(* CoDeSys 2.3.9.45 project: Ascenseur_Augustin_FUCHS.pro *)
(* Libraries: standard.lib 2.6.14 10:37:46, Util.lib 26.9.14 10:12:46 *)

(* Global variable list: Variables_Globales *)
VAR_GLOBAL
(* ----------------------------------
	Entrée
-------------------------------------*)
	(*Présence étage*)
	PRDC: BOOL;
	PET1: BOOL;
	PET2: BOOL;
	PET3: BOOL;

	(*Appel à partir du palier de l'étage*)
	PALRDC: BOOL;
	PALD1: BOOL;
	PALM1: BOOL;
	PALD2: BOOL;
	PALM2: BOOL;
	PAL3: BOOL;

	(*Clignotement d'Appel à partir du palier de l'étage*)
	PALRDCcligno: BOOL;
	PALD1cligno: BOOL;
	PALM1cligno: BOOL;
	PALD2cligno: BOOL;
	PALM2cligno: BOOL;
	PAL3cligno: BOOL;

	(*Appel à partir de la cabine*)
	CABRDC: BOOL;
	CABET1: BOOL;
	CABET2: BOOL;
	CABET3: BOOL;

	(*Porte fermée*)
	PRDCouv: BOOL;
	P1ouv: BOOL;
	P2ouv: BOOL;
	P3ouv: BOOL;

	(*Porte ouverte*)
	PRDCfer: BOOL;
	P1fer: BOOL;
	P2fer: BOOL;
	P3fer: BOOL;

	(* Obstacle a la fermeture*)
	Obs: BOOL;

	(* Arret dy systeme *)
(* ----------------------------------
	Sorties
-------------------------------------*)
	(*Ouverture de porte*)
	ORDC: BOOL;
	O1: BOOL;
	O2: BOOL;
	O3: BOOL;

	(*Fermeture de porte*)
	FRDC: BOOL;
	F1: BOOL;
	F2: BOOL;
	F3: BOOL;

	(*Moteur cabine*)
	CABD: BOOL;
	CABM: BOOL;

	(*Voyant de présence d'étage*)
	VPALRDC: BOOL;
	VPAL1: BOOL;
	VPAL2: BOOL;
	VPAL3: BOOL;

	(*Voyant d'apple étage*)
	VRDC: BOOL;
	V1: BOOL;
	V2: BOOL;
	V3: BOOL;

(* ----------------------------------
		Autres Variables
-------------------------------------*)
	(*Variable du Timer*)
	T1: TP;
	(*Variable d'initialization*)
	STOPbuttonVar: BOOL;
	CABDstatus: BOOL;
	CABMstatus: BOOL;
	T2: TP;
	ESTINIT2: BOOL;
	ReinitAscenseur: BOOL;
	SFCInit: BOOL;
	SFCReset: BOOL;
	T3: TP;
	COUNTSTEP: INT;
	CompteurFor: INT;
	ETAGE_SUIVANT: INT;
	SENS_M: BOOL;
	TableDeVeriteMontee: ARRAY [1..4] OF BOOL;
	TableDeVeriteDesc: ARRAY [1..4] OF BOOL;
	TestSens: INT;
	PROCHAIN_ARRET: INT;
	ArretsDesc: ARRAY [1..4] OF INT;
	ArretsMonte: ARRAY [1..4] OF INT;
	RE_OUVRE: BOOL;
	ARRETcabRDC: BOOL;
	ARRETcabM1: BOOL;
	ARRETcabD1: BOOL;
	ARRETcabM2: BOOL;
	ARRETcabD2: BOOL;
	ARRETcabET3: BOOL;
	CABRDCswitch: BOOL;
	CABET1switch: BOOL;
	CABET2switch: BOOL;
	CABET3switch: BOOL;

	UpFleche: BOOL;
	DownFleche: BOOL;
	RightFleche: BOOL;
	LeftFleche: BOOL;
	FlecheSwitch:BOOL;

	CABmoveY: INT;
	VisuRDCDx: INT;
	VisuRDCDy: REAL;
	VisuRDCGx: REAL;
	VisuRDCGy: REAL;
	VisuET1Dx: INT;
	VisuET1Dy: REAL;
	VisuET1Gx: REAL;
	VisuET1Gy:REAL;
	VisuET2Dx: INT;
	VisuET2Dy: REAL;
	VisuET2Gx: REAL;
	VisuET2Gy: REAL;
	VisuET3Dx: INT;
	VisuET3Dy: REAL;
	VisuET3Gx: REAL;
	VisuET3Gy: REAL;
	InitPortesAscSalon: BOOL;
	T6: TP;
	TIMEURblock: BOOL;
	CompteActionsTime: INT;
	wait: TP;
	PALRDCsave: BOOL;
	PALD1save: BOOL;
	PALM1save: BOOL;
	PALD2save: BOOL;
	PALM2save: BOOL;
	PAL3save: BOOL;
	CABRDCsave: BOOL;
	CABET1save: BOOL;
	CABET2save: BOOL;
	CABET3save: BOOL;
	AfficheBoutonsReset: BOOL;
	BoutonResetVrai: BOOL;
	BoutonRepriseVrai: BOOL;
	STOPbuttonVarImpuls: BOOL;
	ARRETcabRDCsave: BOOL;
	ARRETcabM1save: BOOL;
	ARRETcabD1save: BOOL;
	ARRETcabM2save: BOOL;
	ARRETcabD2save: BOOL;
	ARRETcabET3save: BOOL;
	ReOuvreCabine: BOOL;
	ForceFermeCabine: BOOL;
	BoutonRepriseStopSwitch: BOOL;
	ZoneDepCab: INT;
	DisplayNumbET3: BOOL;
	DisplayNumbET2: BOOL;
	DisplayNumbET1: BOOL;
	DisplayNumbETRDC: BOOL;
	FLECHE_VERS: BOOL;
	DisplayVersRDC: BOOL;
	DisplayVersET1: BOOL;
	DisplayVersET2: BOOL;
	DisplayVersET3: BOOL;
	FinDefinition_SENS: BOOL;
	Offset_ChiffreY: INT;
	CABDsave: BOOL;
	CABMsave: BOOL;
	ORDCsave: BOOL;
	O1save: BOOL;
	O2save: BOOL;
	O3save: BOOL;
	F1save: BOOL;
	FRDCsave: BOOL;
	F2save: BOOL;
	F3save: BOOL;
	PROCHAIN_ARRETsave: INT;
	ETAGE_SUIVANTsave: INT;
	AfficheBoutonsReset2: BOOL;
	StanbyActive: BOOL;
	EXIT_StanbyFunc: BOOL;
	Niveau_Actuel: INT;
	Ancien_Niveau: INT;
	Last_Capt_Pres_Rec: INT;
END_VAR

(* POU PLC_PRG, SFC *)
PROGRAM PLC_PRG
VAR
END_VAR
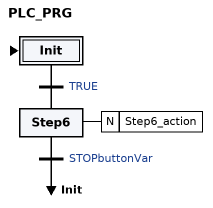
INITIAL_STEP Init:
END_STEP
TRANSITION FROM Init TO Step6 := TRUE;
END_TRANSITION
STEP Step6:
	Step6_action(N);
END_STEP
TRANSITION FROM Step6 TO Init := STOPbuttonVar;
END_TRANSITION

ACTION Step6_action:
PRG_MAIN;
Quel_Etage();
Priorite_Memo();
Appel_Palier();
Arret_Urgence();
ZAuto_RUN();
END_ACTION
END_PROGRAM

(* POU PRG_MAIN, SFC *)
PROGRAM PRG_MAIN
VAR
END_VAR
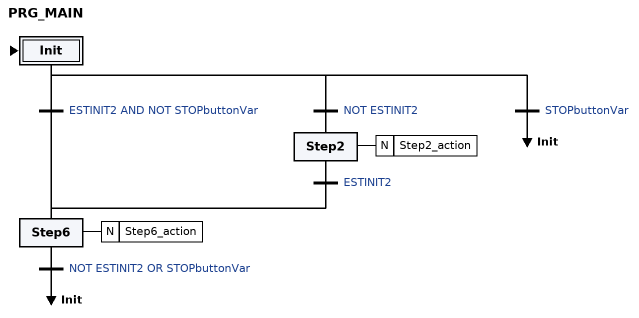
INITIAL_STEP Init:
END_STEP
TRANSITION FROM Init TO Step6 := ESTINIT2 AND NOT STOPbuttonVar;
END_TRANSITION
TRANSITION FROM Init TO Step2 := NOT ESTINIT2;
END_TRANSITION
TRANSITION FROM Init TO Init := STOPbuttonVar;
END_TRANSITION
STEP Step2:
	Step2_action(N);
END_STEP
TRANSITION FROM Step2 TO Step6 := ESTINIT2;
END_TRANSITION
STEP Step6:
	Step6_action(N);
END_STEP
TRANSITION FROM Step6 TO Init := NOT ESTINIT2 OR STOPbuttonVar;
END_TRANSITION

ACTION Step2_action:
IF StanbyActive THEN Correspondance_Etages ();END_IF
Initialisation_reset();
SENS_M:=TRUE;
END_ACTION

ACTION Step6_action:
PAL_COMMUN_ETAGE;
StandBY;
Clignotement;
STOP_PORTES();
Correspondance_Etages();
END_ACTION
END_PROGRAM

(* POU Fonctions_Usuelles/Correspondance_Etages, ST *)
FUNCTION Correspondance_Etages : BOOL
VAR_INPUT
END_VAR
VAR
	CabPosBout: INT;
	PosAscActu: INT;
END_VAR
(*
	Cette fonction à pour but de faire correspondre un appui de la cabine à un appel provenant du palier (sans activer de bouton)
	le but étant de limiter les variables et de se caller sur le cycle existant fonctionnel

	Après avoir récuperer la position de l'ascenseur, nous allons faire correspondre le sens pour que l'étage demandé soit e porchain deservie (dans le cycle)

	Si l'etage demandé est dans le sens et n'as pas encore été demandé, alors il sera dans ce sens
	Si l'étage demandé est déja passé alors nous nous callons sur l'autre sens pour qu'il soit deservie au porchain cycle
*)

PosAscActu:= Last_Capt_Pres();
IF CABRDCswitch THEN
	IF NOT ARRETcabRDC THEN ARRETcabRDC:=TRUE;END_IF
	CABRDC:=TRUE;
END_IF

IF CABET1switch THEN
	CabPosBout:=2;
	IF PosAscActu < 5 OR  ETAGE_SUIVANT < 9 THEN
		IF PosAscActu >= 5 THEN PosAscActu:= ETAGE_SUIVANT;END_IF
 		IF SENS_M THEN
			IF PosAscActu <= CabPosBout THEN ARRETcabM1:=TRUE;
			ELSE ARRETcabD1:=TRUE;END_IF
		ELSE
			IF PosAscActu >= CabPosBout THEN ARRETcabD1:=TRUE;
			ELSE ARRETcabM1:=TRUE;END_IF
		END_IF
	ELSE
		IF SENS_M THEN
			IF NOT ARRETcabM1 THEN ARRETcabM1:=TRUE;END_IF
		ELSE
			IF NOT ARRETcabD1 THEN ARRETcabD1:=TRUE;END_IF
		END_IF
	END_IF
	CABET1:=TRUE;
END_IF

IF CABET2switch THEN
	CabPosBout:=3;
	IF PosAscActu < 5 OR  ETAGE_SUIVANT < 9 THEN
		IF PosAscActu >= 5 THEN PosAscActu:= ETAGE_SUIVANT;END_IF
 		IF SENS_M THEN
			IF PosAscActu <= CabPosBout THEN ARRETcabM2:=TRUE;
			ELSE ARRETcabD2:=TRUE;END_IF
		ELSE
			IF PosAscActu >= CabPosBout THEN ARRETcabD2:=TRUE;
			ELSE ARRETcabM2:=TRUE;END_IF
		END_IF
	ELSE
		IF SENS_M THEN
			IF NOT ARRETcabM2 THEN ARRETcabM2:=TRUE;END_IF
		ELSE
			IF NOT ARRETcabD2 THEN ARRETcabD2:=TRUE;END_IF
		END_IF
	END_IF
	CABET2:=TRUE;
END_IF

IF CABET3switch THEN
	CabPosBout:=4;
	IF NOT ARRETcabET3 THEN ARRETcabET3:=TRUE;END_IF
	CABET3:=TRUE;
END_IF

(*Si un appel palier est effectué, il est associé à sa mémorisation*)
IF PALRDC THEN ARRETcabRDC:=TRUE;END_IF
IF PALD1 THEN ARRETcabD1:=TRUE;END_IF
IF PALM1 THEN ARRETcabM1:=TRUE;END_IF
IF PALD2 THEN ARRETcabD2:=TRUE;END_IF
IF PALM2 THEN ARRETcabM2:=TRUE;END_IF
IF PAL3 THEN ARRETcabET3:=TRUE;END_IF
END_FUNCTION

(* POU Fonctions_Usuelles/Last_Capt_Pres, ST *)
FUNCTION Last_Capt_Pres : INT
VAR_INPUT
END_VAR
VAR
END_VAR
(*cette fonction se rapproche de get_floor mais elle permet d'obtenir le dernier capteur ou était l'ascenseur*)
IF PRDC=TRUE THEN Last_Capt_Pres_Rec:=1;
ELSIF PET1=TRUE THEN Last_Capt_Pres_Rec:=2;
ELSIF PET2=TRUE THEN Last_Capt_Pres_Rec:=3;
ELSIF PET3=TRUE THEN Last_Capt_Pres_Rec:=4; END_IF
IF NOT PRDC AND NOT PET1 AND NOT PET2 AND NOT PET3 THEN
	Last_Capt_Pres:=Last_Capt_Pres_Rec;
	IF CABM AND NOT CABD THEN
		Last_Capt_Pres:= Last_Capt_Pres_Rec+1;
	ELSIF CABD AND NOT CABM THEN
		Last_Capt_Pres:= Last_Capt_Pres_Rec-1;
	END_IF
	IF Last_Capt_Pres > 4 THEN Last_Capt_Pres:=4;END_IF
	IF Last_Capt_Pres = 0 THEN Last_Capt_Pres:=1;END_IF
ELSE
	Last_Capt_Pres:=Last_Capt_Pres_Rec;
END_IF
END_FUNCTION

(* POU PAL_COMMUN_ETAGE, SFC *)
PROGRAM PAL_COMMUN_ETAGE
VAR
	ARRET_EN_COURS: INT;
	ATTEND_UN_PEU: BOOL;
	T5: TP;
END_VAR
(*AND ETAGE_SUIVANT = 2 AND NOT SENS_M*)
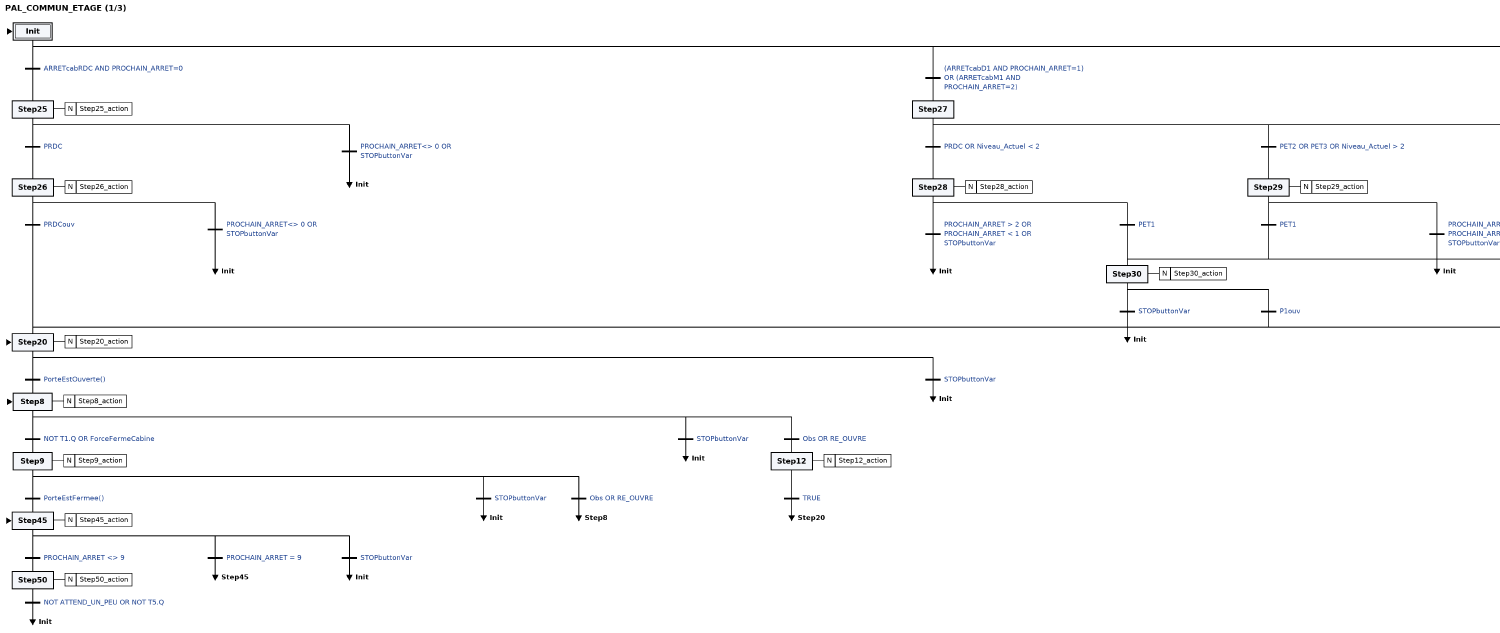
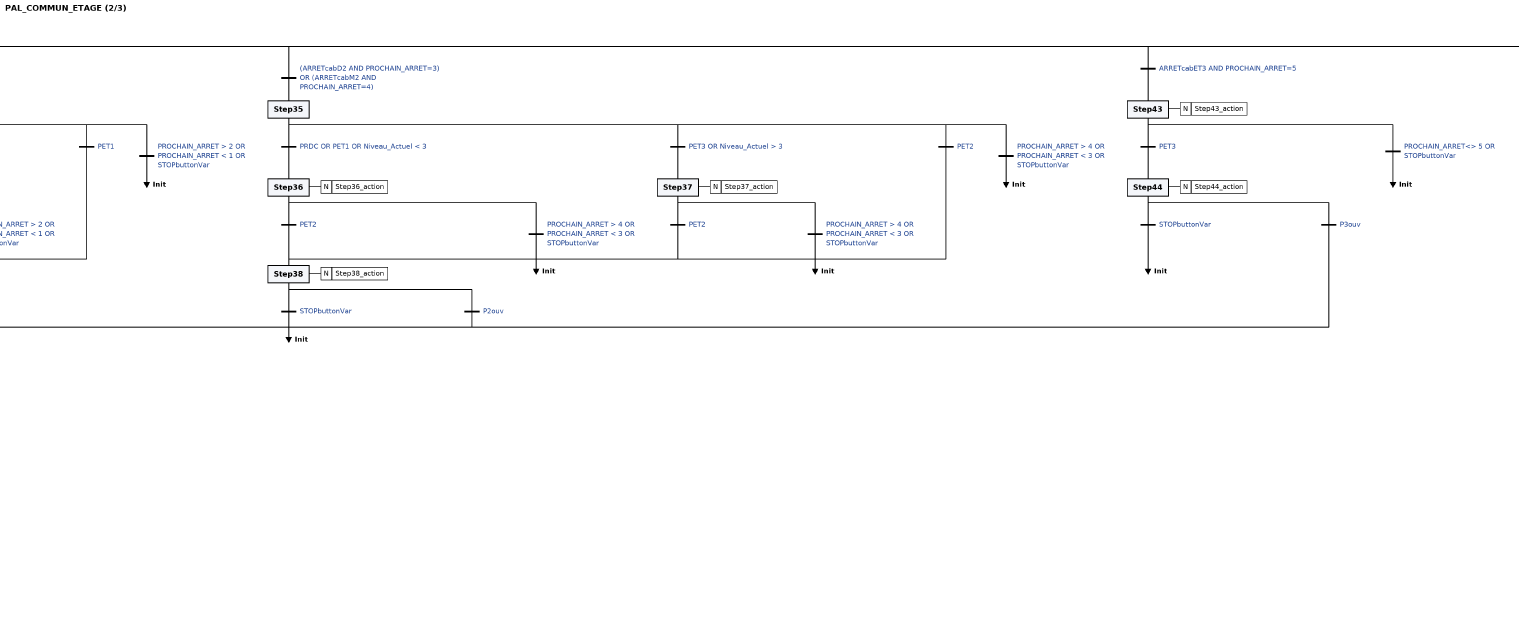
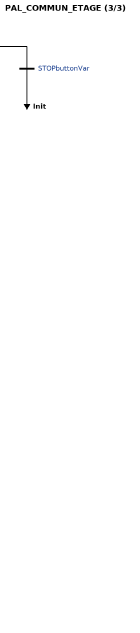
INITIAL_STEP Init:
END_STEP
TRANSITION FROM Init TO Step25 := ARRETcabRDC AND PROCHAIN_ARRET=0;
END_TRANSITION
TRANSITION FROM Init TO Step27 := (ARRETcabD1 AND PROCHAIN_ARRET=1) OR (ARRETcabM1 AND PROCHAIN_ARRET=2);
END_TRANSITION
TRANSITION FROM Init TO Step35 := (ARRETcabD2 AND PROCHAIN_ARRET=3) OR (ARRETcabM2 AND PROCHAIN_ARRET=4);
END_TRANSITION
TRANSITION FROM Init TO Step43 := ARRETcabET3 AND PROCHAIN_ARRET=5;
END_TRANSITION
TRANSITION FROM Init TO Init := STOPbuttonVar;
END_TRANSITION
STEP Step25:
	Step25_action(N);
END_STEP
TRANSITION FROM Step25 TO Step26 := PRDC;
END_TRANSITION
TRANSITION FROM Step25 TO Init := PROCHAIN_ARRET<> 0 OR STOPbuttonVar;
END_TRANSITION
STEP Step26:
	Step26_action(N);
END_STEP
TRANSITION FROM Step26 TO Step20 := PRDCouv;
END_TRANSITION
TRANSITION FROM Step26 TO Init := PROCHAIN_ARRET<> 0 OR STOPbuttonVar;
END_TRANSITION
STEP Step27:
END_STEP
TRANSITION FROM Step27 TO Step28 := PRDC OR Niveau_Actuel < 2;
END_TRANSITION
TRANSITION FROM Step27 TO Step29 := PET2 OR PET3 OR Niveau_Actuel > 2;
END_TRANSITION
TRANSITION FROM Step27 TO Step30 := PET1;
END_TRANSITION
TRANSITION FROM Step27 TO Init := PROCHAIN_ARRET > 2 OR PROCHAIN_ARRET < 1 OR  STOPbuttonVar;
END_TRANSITION
STEP Step28:
	Step28_action(N);
END_STEP
TRANSITION FROM Step28 TO Init := PROCHAIN_ARRET > 2 OR PROCHAIN_ARRET < 1 OR  STOPbuttonVar;
END_TRANSITION
TRANSITION FROM Step28 TO Step30 := PET1;
END_TRANSITION
STEP Step29:
	Step29_action(N);
END_STEP
TRANSITION FROM Step29 TO Step30 := PET1;
END_TRANSITION
TRANSITION FROM Step29 TO Init := PROCHAIN_ARRET > 2 OR PROCHAIN_ARRET < 1 OR  STOPbuttonVar;
END_TRANSITION
STEP Step30:
	Step30_action(N);
END_STEP
TRANSITION FROM Step30 TO Init := STOPbuttonVar;
END_TRANSITION
TRANSITION FROM Step30 TO Step20 := P1ouv;
END_TRANSITION
STEP Step35:
END_STEP
TRANSITION FROM Step35 TO Step36 := PRDC OR PET1 OR Niveau_Actuel < 3;
END_TRANSITION
TRANSITION FROM Step35 TO Step37 := PET3 OR Niveau_Actuel > 3;
END_TRANSITION
TRANSITION FROM Step35 TO Step38 := PET2;
END_TRANSITION
TRANSITION FROM Step35 TO Init := PROCHAIN_ARRET > 4 OR PROCHAIN_ARRET < 3 OR  STOPbuttonVar;
END_TRANSITION
STEP Step36:
	Step36_action(N);
END_STEP
TRANSITION FROM Step36 TO Step38 := PET2;
END_TRANSITION
TRANSITION FROM Step36 TO Init := PROCHAIN_ARRET > 4 OR PROCHAIN_ARRET < 3 OR  STOPbuttonVar;
END_TRANSITION
STEP Step37:
	Step37_action(N);
END_STEP
TRANSITION FROM Step37 TO Step38 := PET2;
END_TRANSITION
TRANSITION FROM Step37 TO Init := PROCHAIN_ARRET > 4 OR PROCHAIN_ARRET < 3 OR  STOPbuttonVar;
END_TRANSITION
STEP Step38:
	Step38_action(N);
END_STEP
TRANSITION FROM Step38 TO Init := STOPbuttonVar;
END_TRANSITION
TRANSITION FROM Step38 TO Step20 := P2ouv;
END_TRANSITION
STEP Step43:
	Step43_action(N);
END_STEP
TRANSITION FROM Step43 TO Step44 := PET3;
END_TRANSITION
TRANSITION FROM Step43 TO Init := PROCHAIN_ARRET<> 5 OR STOPbuttonVar;
END_TRANSITION
STEP Step44:
	Step44_action(N);
END_STEP
TRANSITION FROM Step44 TO Init := STOPbuttonVar;
END_TRANSITION
TRANSITION FROM Step44 TO Step20 := P3ouv;
END_TRANSITION
STEP Step20:
	Step20_action(N);
END_STEP
TRANSITION FROM Step20 TO Step8 := PorteEstOuverte();
END_TRANSITION
TRANSITION FROM Step20 TO Init := STOPbuttonVar;
END_TRANSITION
STEP Step8:
	Step8_action(N);
END_STEP
TRANSITION FROM Step8 TO Step9 := NOT T1.Q OR ForceFermeCabine;
END_TRANSITION
TRANSITION FROM Step8 TO Init := STOPbuttonVar;
END_TRANSITION
TRANSITION FROM Step8 TO Step12 := Obs OR RE_OUVRE;
END_TRANSITION
STEP Step12:
	Step12_action(N);
END_STEP
TRANSITION FROM Step12 TO Step20 := TRUE;
END_TRANSITION
STEP Step9:
	Step9_action(N);
END_STEP
TRANSITION FROM Step9 TO Step45 := PorteEstFermee();
END_TRANSITION
TRANSITION FROM Step9 TO Init := STOPbuttonVar;
END_TRANSITION
TRANSITION FROM Step9 TO Step8 := Obs OR RE_OUVRE;
END_TRANSITION
STEP Step45:
	Step45_action(N);
END_STEP
TRANSITION FROM Step45 TO Step50 := PROCHAIN_ARRET <> 9;
END_TRANSITION
TRANSITION FROM Step45 TO Step45 := PROCHAIN_ARRET = 9;
END_TRANSITION
TRANSITION FROM Step45 TO Init := STOPbuttonVar;
END_TRANSITION
STEP Step50:
	Step50_action(N);
END_STEP
TRANSITION FROM Step50 TO Init := NOT ATTEND_UN_PEU OR NOT T5.Q;
END_TRANSITION

ACTION Step25_action:
CABD:=TRUE;
CABM:=FALSE;
END_ACTION

ACTION Step26_action:
CABD:=FALSE;
ORDC:=TRUE;
CABRDC:=FALSE;
ARRET_EN_COURS:=PROCHAIN_ARRET;
Reset_Arrets_CAB(ARRET_EN_COURS);
END_ACTION

ACTION Step28_action:
CABM:=TRUE;
CABD:=FALSE;
END_ACTION

ACTION Step29_action:
CABD:=TRUE;
CABM:=FALSE;
END_ACTION

ACTION Step30_action:
ARRET_EN_COURS:=PROCHAIN_ARRET;
CABM:=FALSE;
CABD:=FALSE;
O1:=TRUE;
CABET1:=FALSE;
Reset_Arrets_CAB(ARRET_EN_COURS);
END_ACTION

ACTION Step36_action:
CABM:=TRUE;
CABD:=FALSE;
END_ACTION

ACTION Step37_action:
CABD:=TRUE;
CABM:=FALSE;
END_ACTION

ACTION Step38_action:
ARRET_EN_COURS:=PROCHAIN_ARRET;
CABM:=FALSE;
CABD:=FALSE;
O2:=TRUE;
CABET2:=FALSE;
Reset_Arrets_CAB(ARRET_EN_COURS);
END_ACTION

ACTION Step43_action:
CABM:=TRUE;
CABD:=FALSE;
END_ACTION

ACTION Step44_action:
CABM:=FALSE;
O3:=TRUE;
CABET3:=FALSE;
ARRET_EN_COURS:=PROCHAIN_ARRET;
Reset_Arrets_CAB(ARRET_EN_COURS);
END_ACTION

ACTION Step20_action:
T1(IN:=FALSE);
RE_OUVRE:=FALSE;
END_ACTION

ACTION Step8_action:
(*Switch Button
IF P1fer THEN P1fer:=FALSE;
END_IF;
*)
ORDC:=FALSE;
O1:=FALSE;
O2:=FALSE;
O3:=FALSE;
T1(IN:=TRUE, PT:=t#2s);
Re_ouverture();
END_ACTION

ACTION Step12_action:
IF NOT PorteEstOuverte() THEN Ouv_Fer_Etage(TRUE);
END_IF
FRDC:=FALSE;
F1:=FALSE;
F2:=FALSE;
F3:=FALSE;
T1(IN:=FALSE);
T1(IN:=TRUE, PT:=t#1ms);
RE_OUVRE:=FALSE;
END_ACTION

ACTION Step9_action:
(*IF NOT Obs THEN F1:=TRUE;*)
Re_ouverture();
IF NOT Obs THEN
	Ouv_Fer_Etage(FALSE);
END_IF
T1(IN:=FALSE);
T5(IN:=FALSE);
END_ACTION

ACTION Step45_action:
(* Switch Button
IF P1ouv THEN P1ouv:=FALSE;
END_IF*)
FRDC:=FALSE;
F1:=FALSE;
F2:=FALSE;
F3:=FALSE;
RE_OUVRE:=FALSE;
IF PROCHAIN_ARRET <>  9 THEN Reset_Arrets(ARRET_EN_COURS);END_IF
END_ACTION

ACTION Step50_action:
(*Fonction pour l'attente d'appel dans la cabien avant un changelent de sens*)

ATTEND_UN_PEU:=FALSE;
IF PROCHAIN_ARRET <> 0 AND PROCHAIN_ARRET <> 5 THEN
	IF PROCHAIN_ARRET = ARRET_EN_COURS THEN
		ATTEND_UN_PEU:=TRUE;
	ELSE
		IF PROCHAIN_ARRET - ARRET_EN_COURS = 1 OR ARRET_EN_COURS - PROCHAIN_ARRET = 1 THEN
			IF PROCHAIN_ARRET MOD 2 = 1 THEN
				IF PROCHAIN_ARRET < ARRET_EN_COURS THEN ATTEND_UN_PEU:=TRUE;END_IF
			ELSE
				IF PROCHAIN_ARRET > ARRET_EN_COURS THEN ATTEND_UN_PEU:=TRUE;END_IF
			END_IF
		END_IF
	END_IF
END_IF
T5(IN:=TRUE,PT:=t#5s);

IF ATTEND_UN_PEU THEN
	ETAGE_SUIVANT:=9;
	PROCHAIN_ARRET:=9;
	IF ARRET_EN_COURS MOD 2 = 1 THEN SENS_M:=FALSE;
	ELSE SENS_M:=TRUE;END_IF
END_IF
END_ACTION
END_PROGRAM

(* POU Fonctions_Usuelles/Capteurs/PorteEstOuverte, ST *)
FUNCTION PorteEstOuverte : BOOL
VAR_INPUT
END_VAR
VAR
END_VAR
(*Cette fonction permet de savoir si la porte à l'étage ou se trouve l'ascenseur est ouverte.
Elle renvoie true si elle est ouverte.
*)
PorteEstOuverte:=FALSE;
IF Get_Floor() = 0 THEN
	IF PRDCouv THEN PorteEstOuverte:=TRUE;
	ELSE PorteEstOuverte:=FALSE;
	END_IF
ELSIF Get_Floor() = 1 THEN
	IF P1ouv  THEN PorteEstOuverte:=TRUE;
	ELSE PorteEstOuverte:=FALSE;
	END_IF
ELSIF Get_Floor() = 2 THEN
	IF P2ouv  THEN PorteEstOuverte:=TRUE;
	ELSE PorteEstOuverte:=FALSE;
	END_IF
ELSIF Get_Floor() = 3 THEN
	IF P3ouv  THEN PorteEstOuverte:=TRUE;
	ELSE PorteEstOuverte:=FALSE;
	END_IF
END_IF
END_FUNCTION

(* POU Fonctions_Usuelles/Capteurs/Get_Floor, ST *)
FUNCTION Get_Floor : INT
VAR_INPUT
END_VAR
VAR
END_VAR
(*
Cette fonction renvoie l'étage de l'ascenseur si il est arreté à un étage
renvoie une valeur supérieur si il est en mouvement
*)
IF PRDC=TRUE THEN Get_Floor:=0;
ELSIF PET1=TRUE THEN Get_Floor:=1;
ELSIF PET2=TRUE THEN Get_Floor:=2;
ELSIF PET3=TRUE THEN Get_Floor:=3;
ELSE Get_Floor:=4;
END_IF
(*0n verifie que l'ascenceur n'est pas en cours de mouvement*)
IF CABD OR CABM THEN Get_Floor:=5;END_IF
END_FUNCTION

(* POU Fonctions_Usuelles/Ouv_Fer_Etage, ST *)
FUNCTION Ouv_Fer_Etage : BOOL
VAR_INPUT
	(*True pour ouvrir et False pour fermer*)
	OuvrirFermer:BOOL;
END_VAR
VAR
END_VAR
(*Cette fonction ouvre la porte de l'étage à laquelle il se trouve l'ascenseur si ell est vrai
la ferme si elle est fausse*)
IF OuvrirFermer THEN
	IF Get_Floor() = 0 THEN
		IF NOT PRDCouv THEN ORDC:=TRUE;END_IF
	ELSIF Get_Floor() = 1 THEN
		IF NOT P1ouv THEN O1:=TRUE;END_IF
	ELSIF Get_Floor() = 2 THEN
		IF NOT P2ouv THEN O2:=TRUE;END_IF
	ELSIF Get_Floor() = 3 THEN
		IF NOT P3ouv THEN O3:=TRUE;END_IF
	END_IF
ELSE
	IF Get_Floor() = 0 THEN
		IF NOT PRDCfer THEN FRDC:=TRUE;END_IF
	ELSIF Get_Floor() = 1 THEN
		IF NOT P1fer THEN F1:=TRUE;END_IF
	ELSIF Get_Floor() = 2 THEN
		IF NOT P2fer THEN F2:=TRUE;END_IF
	ELSIF Get_Floor() = 3 THEN
		IF NOT P3fer THEN F3:=TRUE;END_IF
	END_IF
END_IF
END_FUNCTION

(* POU Fonctions_Usuelles/Capteurs/PorteEstFermee, ST *)
FUNCTION PorteEstFermee : BOOL
VAR_INPUT
END_VAR
VAR
END_VAR
(*Cette fonction permet de savoir si la porte à l'étage ou se trouve l'ascenseur est fermée.
Elle renvoie true si elle est fermée.
*)
PorteEstFermee:=FALSE;
IF Get_Floor() = 0 THEN
	IF PRDCfer THEN PorteEstFermee:=TRUE;
	ELSE PorteEstFermee:=FALSE;
	END_IF
ELSIF Get_Floor() = 1 THEN
	IF P1fer  THEN PorteEstFermee:=TRUE;
	ELSE PorteEstFermee:=FALSE;
	END_IF
ELSIF Get_Floor() = 2 THEN
	IF P2fer  THEN PorteEstFermee:=TRUE;
	ELSE PorteEstFermee:=FALSE;
	END_IF
ELSIF Get_Floor() = 3 THEN
	IF P3fer  THEN PorteEstFermee:=TRUE;
	ELSE PorteEstFermee:=FALSE;
	END_IF
END_IF
END_FUNCTION

(* POU Fonctions_Usuelles/Voyants_boutons/Reset_Arrets, ST *)
FUNCTION Reset_Arrets : BOOL
VAR_INPUT
	ARRET_EN_COURS: INT;
END_VAR
VAR
END_VAR
(* cette fonction permet de réinitialiser tout les arrets d'un étage pour permettre un nouvel appel lors d'un prochain cycle*)
IF ARRET_EN_COURS=0 THEN
	PALRDC:=FALSE;
	CABRDC:=FALSE;
	ARRETcabRDC:=FALSE;
ELSIF ARRET_EN_COURS=1 THEN
	PALD1:=FALSE;
	CABET1:=FALSE;
	ARRETcabD1:=FALSE;
ELSIF ARRET_EN_COURS=2 THEN
	PALM1:=FALSE;
	CABET1:=FALSE;
	ARRETcabM1:=FALSE;
ELSIF ARRET_EN_COURS=3 THEN
	PALD2:=FALSE;
	CABET2:=FALSE;
	ARRETcabD2:=FALSE;
ELSIF ARRET_EN_COURS=4 THEN
	ARRETcabM2:=FALSE;
	PALM2:=FALSE;
	CABET2:=FALSE;
ELSIF ARRET_EN_COURS=5 THEN
	PAL3:=FALSE;
	CABET3:=FALSE;
	ARRETcabET3:=FALSE;
END_IF
ETAGE_SUIVANT:=9;
END_FUNCTION

(* POU Fonctions_Usuelles/Voyants_boutons/Clignotement, SFC *)
PROGRAM Clignotement
VAR
END_VAR
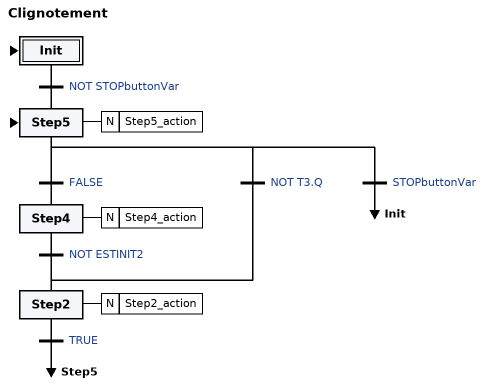
INITIAL_STEP Init:
END_STEP
TRANSITION FROM Init TO Step5 := NOT STOPbuttonVar;
END_TRANSITION
STEP Step5:
	Step5_action(N);
END_STEP
TRANSITION FROM Step5 TO Step4 := FALSE;
END_TRANSITION
TRANSITION FROM Step5 TO Step2 := NOT T3.Q;
END_TRANSITION
TRANSITION FROM Step5 TO Init := STOPbuttonVar;
END_TRANSITION
STEP Step4:
	Step4_action(N);
END_STEP
TRANSITION FROM Step4 TO Step2 := NOT ESTINIT2;
END_TRANSITION
STEP Step2:
	Step2_action(N);
END_STEP
TRANSITION FROM Step2 TO Step5 := TRUE;
END_TRANSITION

ACTION Step5_action:
T3(IN:=TRUE, PT:=t#500ms);
END_ACTION

ACTION Step4_action:
T2(IN:=FALSE);
ESTINIT2:=FALSE;
END_ACTION

ACTION Step2_action:
(* IF  CABD OR CABM OR ORDC OR O1 OR O2 OR O3 OR NOT PRDCfer OR NOT P1fer OR NOT P2fer OR NOT P3fer OR PAL3 OR PALM2 OR  PALD2 OR PALD1 OR PALM1 OR PALRDC THEN
	T2(IN:=TRUE, PT:=t#10s);
ELSE
	T2(IN:=FALSE);
END_IF
*)
IF PALRDC THEN
	IF VRDC THEN VRDC:=FALSE;
	ELSE VRDC:=TRUE;END_IF
END_IF
IF PALD1 OR PALM1 THEN
	IF V1 THEN V1:=FALSE;
	ELSE V1:=TRUE;END_IF
END_IF
IF PALD2 OR PALM2 THEN
	IF V2 THEN V2:=FALSE;
	ELSE V2:=TRUE;END_IF
END_IF
IF PAL3 THEN
	IF V3 THEN V3:=FALSE;
	ELSE V3:=TRUE;END_IF
END_IF
T3(IN:=FALSE);
T3(IN:=TRUE, PT:=t#1ms);
END_ACTION
END_PROGRAM

(* POU Initialisation_Standby/ETAGE_1, SFC *)
PROGRAM ETAGE_1
VAR
END_VAR
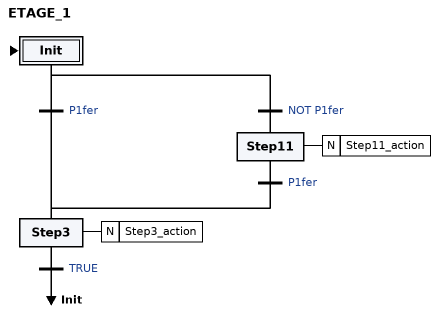
INITIAL_STEP Init:
END_STEP
TRANSITION FROM Init TO Step3 := P1fer;
END_TRANSITION
TRANSITION FROM Init TO Step11 := NOT P1fer;
END_TRANSITION
STEP Step11:
	Step11_action(N);
END_STEP
TRANSITION FROM Step11 TO Step3 := P1fer;
END_TRANSITION
STEP Step3:
	Step3_action(N);
END_STEP
TRANSITION FROM Step3 TO Init := TRUE;
END_TRANSITION

ACTION Step11_action:
F1:=TRUE;
END_ACTION

ACTION Step3_action:
F1:=FALSE;
END_ACTION
END_PROGRAM

(* POU Initialisation_Standby/ETAGE_2, SFC *)
PROGRAM ETAGE_2
VAR
END_VAR
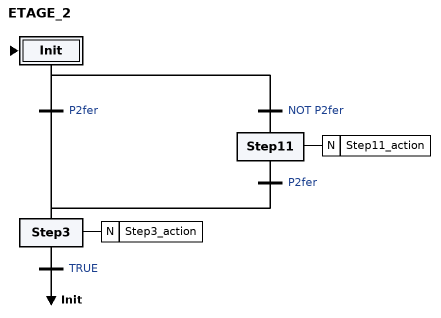
INITIAL_STEP Init:
END_STEP
TRANSITION FROM Init TO Step3 := P2fer;
END_TRANSITION
TRANSITION FROM Init TO Step11 := NOT P2fer;
END_TRANSITION
STEP Step11:
	Step11_action(N);
END_STEP
TRANSITION FROM Step11 TO Step3 := P2fer;
END_TRANSITION
STEP Step3:
	Step3_action(N);
END_STEP
TRANSITION FROM Step3 TO Init := TRUE;
END_TRANSITION

ACTION Step11_action:
F2:=TRUE;
END_ACTION

ACTION Step3_action:
F2:=FALSE;
END_ACTION
END_PROGRAM

(* POU Initialisation_Standby/ETAGE_3, SFC *)
PROGRAM ETAGE_3
VAR
END_VAR
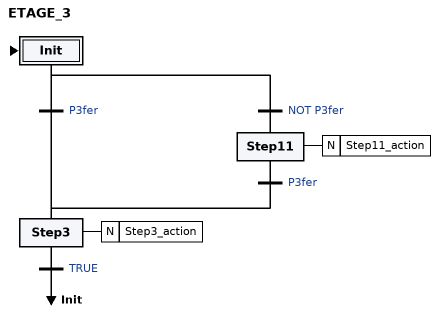
INITIAL_STEP Init:
END_STEP
TRANSITION FROM Init TO Step3 := P3fer;
END_TRANSITION
TRANSITION FROM Init TO Step11 := NOT P3fer;
END_TRANSITION
STEP Step11:
	Step11_action(N);
END_STEP
TRANSITION FROM Step11 TO Step3 := P3fer;
END_TRANSITION
STEP Step3:
	Step3_action(N);
END_STEP
TRANSITION FROM Step3 TO Init := TRUE;
END_TRANSITION

ACTION Step11_action:
F3:=TRUE;
END_ACTION

ACTION Step3_action:
F3:=FALSE;
END_ACTION
END_PROGRAM

(* POU Initialisation_Standby/ETAGE_RDC, SFC *)
PROGRAM ETAGE_RDC
VAR
END_VAR
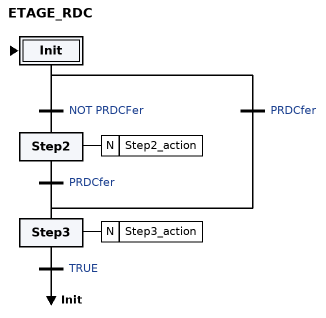
INITIAL_STEP Init:
END_STEP
TRANSITION FROM Init TO Step2 := NOT PRDCFer;
END_TRANSITION
TRANSITION FROM Init TO Step3 := PRDCfer;
END_TRANSITION
STEP Step2:
	Step2_action(N);
END_STEP
TRANSITION FROM Step2 TO Step3 := PRDCfer;
END_TRANSITION
STEP Step3:
	Step3_action(N);
END_STEP
TRANSITION FROM Step3 TO Init := TRUE;
END_TRANSITION

ACTION Step2_action:
FRDC:=TRUE;
END_ACTION

ACTION Step3_action:
FRDC:=FALSE;
Quel_Etage();
END_ACTION
END_PROGRAM

(* POU Initialisation_Standby/Initialisation_reset, SFC *)
PROGRAM Initialisation_reset
VAR
END_VAR
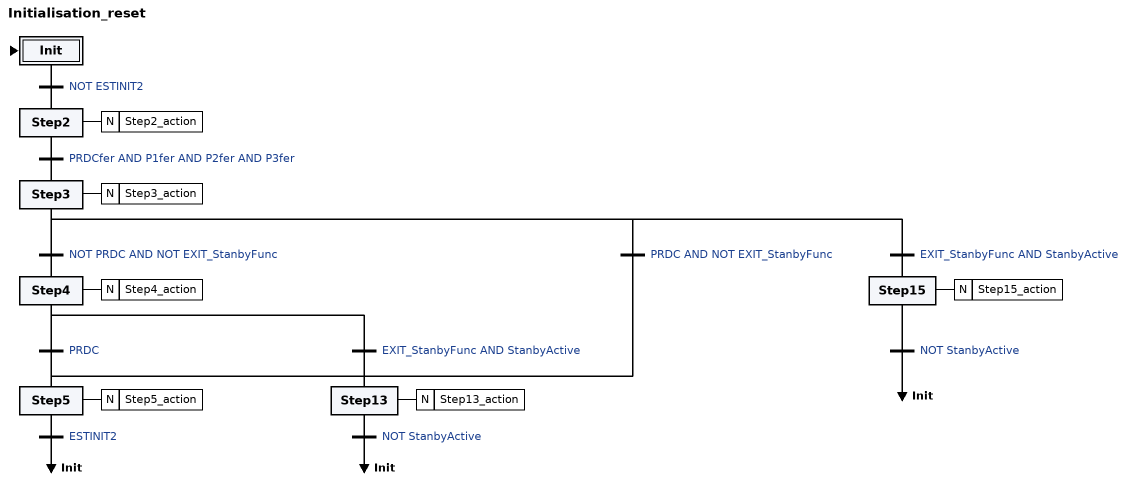
INITIAL_STEP Init:
END_STEP
TRANSITION FROM Init TO Step2 := NOT ESTINIT2;
END_TRANSITION
STEP Step2:
	Step2_action(N);
END_STEP
TRANSITION FROM Step2 TO Step3 := PRDCfer AND P1fer AND P2fer AND P3fer;
END_TRANSITION
STEP Step3:
	Step3_action(N);
END_STEP
TRANSITION FROM Step3 TO Step4 := NOT PRDC AND NOT EXIT_StanbyFunc;
END_TRANSITION
TRANSITION FROM Step3 TO Step5 := PRDC AND NOT EXIT_StanbyFunc;
END_TRANSITION
TRANSITION FROM Step3 TO Step15 := EXIT_StanbyFunc AND StanbyActive;
END_TRANSITION
STEP Step4:
	Step4_action(N);
END_STEP
TRANSITION FROM Step4 TO Step5 := PRDC;
END_TRANSITION
TRANSITION FROM Step4 TO Step13 := EXIT_StanbyFunc AND StanbyActive;
END_TRANSITION
STEP Step13:
	Step13_action(N);
END_STEP
TRANSITION FROM Step13 TO Init := NOT StanbyActive;
END_TRANSITION
STEP Step15:
	Step15_action(N);
END_STEP
TRANSITION FROM Step15 TO Init := NOT StanbyActive;
END_TRANSITION
STEP Step5:
	Step5_action(N);
END_STEP
TRANSITION FROM Step5 TO Init := ESTINIT2;
END_TRANSITION

ACTION Step2_action:
ETAGE_RDC;
ETAGE_1;
ETAGE_2;
ETAGE_3;
ETAGE_SUIVANT:=1;
PROCHAIN_ARRET:=0;
END_ACTION

ACTION Step3_action:
(*Désactivation de tout les moteurs *)
FRDC:=FALSE;
F1:=FALSE;
F2:=FALSE;
F3:=FALSE;
END_ACTION

ACTION Step4_action:
IF NOT PRDC THEN CABD:=TRUE;END_IF
SENS_M:=FALSE;
END_ACTION

ACTION Step13_action:
EXIT_StanbyFunc :=FALSE;
ESTINIT2:=TRUE;
CABD:=FALSE;
ETAGE_SUIVANT:=9;
PROCHAIN_ARRET:=9;
StanbyActive:=FALSE;
END_ACTION

ACTION Step15_action:
EXIT_StanbyFunc:=FALSE;
ESTINIT2:=TRUE;
CABD:=FALSE;
ETAGE_SUIVANT:=9;
PROCHAIN_ARRET:=9;
StanbyActive:=FALSE;
END_ACTION

ACTION Step5_action:
CABD:=FALSE;
ESTINIT2:=TRUE;
StanbyActive:=FALSE;
SENS_M:=TRUE;
ETAGE_SUIVANT:=9;
PROCHAIN_ARRET:=9;
END_ACTION
END_PROGRAM

(* POU Initialisation_Standby/StandBY, SFC *)
PROGRAM StandBY
VAR
END_VAR
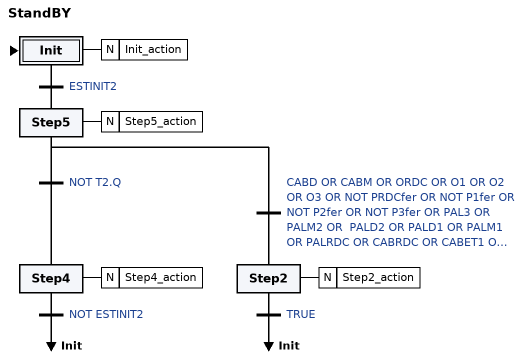
INITIAL_STEP Init:
	Init_action(N);
END_STEP
TRANSITION FROM Init TO Step5 := ESTINIT2;
END_TRANSITION
STEP Step5:
	Step5_action(N);
END_STEP
TRANSITION FROM Step5 TO Step4 := NOT T2.Q;
END_TRANSITION
TRANSITION FROM Step5 TO Step2 := CABD OR CABM OR ORDC OR O1 OR O2 OR O3 OR NOT PRDCfer OR NOT P1fer OR NOT P2fer OR NOT P3fer OR PAL3 OR PALM2 OR  PALD2 OR PALD1 OR PALM1 OR PALRDC OR CABRDC OR CABET1 OR CABET2 OR CABET3;
END_TRANSITION
STEP Step4:
	Step4_action(N);
END_STEP
TRANSITION FROM Step4 TO Init := NOT ESTINIT2;
END_TRANSITION
STEP Step2:
	Step2_action(N);
END_STEP
TRANSITION FROM Step2 TO Init := TRUE;
END_TRANSITION

ACTION Init_action:
T2(IN:=FALSE);
END_ACTION

ACTION Step5_action:
T2(IN:=TRUE, PT:=t#7s);
END_ACTION

ACTION Step4_action:
T2(IN:=FALSE);
ESTINIT2:=FALSE;
StanbyActive:=TRUE;
END_ACTION

ACTION Step2_action:
(* IF  CABD OR CABM OR ORDC OR O1 OR O2 OR O3 OR NOT PRDCfer OR NOT P1fer OR NOT P2fer OR NOT P3fer OR PAL3 OR PALM2 OR  PALD2 OR PALD1 OR PALM1 OR PALRDC THEN
	T2(IN:=TRUE, PT:=t#10s);
ELSE
	T2(IN:=FALSE);
END_IF
*)

T2(IN:=FALSE);
T2(IN:=TRUE, PT:=t#1ms);
END_ACTION
END_PROGRAM

(* POU Simulation_Visuelle/Afficher_Etage_Range, ST *)
FUNCTION Afficher_Etage_Range : BOOL
VAR_INPUT
END_VAR
VAR
END_VAR
(* Cette fonction sert à l'affichage de l'étage dans lequel se trouve l'asenceur,
ainsi que l'étage qui sera desservie prochainement.*)

(* Utilisé uniquement sur la simulation visuelle de l'écran
n'interfère pas avecx le porgramme principal*)

IF 55 < CABmoveY AND CABmoveY<= 110 THEN
	DisplayNumbETRDC:=TRUE;
	DisplayNumbET1:=FALSE;
ELSIF -55 < CABmoveY AND CABmoveY<= 55  THEN
	DisplayNumbET1:=TRUE;
	DisplayNumbETRDC:=FALSE;
	DisplayNumbET2:=FALSE;
ELSIF -165 < CABmoveY AND CABmoveY <= -55  THEN
	DisplayNumbET2:=TRUE;
	DisplayNumbET1:=FALSE;
	DisplayNumbET3:=FALSE;
ELSIF -220 < CABmoveY AND CABmoveY <= -165  THEN
	DisplayNumbET3:=TRUE;
	DisplayNumbET2:=FALSE;
END_IF

IF Get_Floor()+1 <> ETAGE_SUIVANT THEN
	IF ETAGE_SUIVANT =  9 THEN
		FLECHE_VERS:=FALSE;
		DisplayVersRDC:=FALSE;
		DisplayVersET1:=FALSE;
		DisplayVersET2:=FALSE;
		DisplayVersET3:=FALSE;
	ELSIF ETAGE_SUIVANT = 1 THEN
		FLECHE_VERS:=TRUE;
		DisplayVersET1:=FALSE;
		DisplayVersET2:=FALSE;
		DisplayVersET3:=FALSE;
		DisplayVersRDC:=TRUE;
	ELSIF ETAGE_SUIVANT = 2 THEN
		FLECHE_VERS:=TRUE;
		DisplayVersRDC:=FALSE;
		DisplayVersET2:=FALSE;
		DisplayVersET3:=FALSE;
		DisplayVersET1:=TRUE;
	ELSIF ETAGE_SUIVANT = 3 THEN
		FLECHE_VERS:=TRUE;
		DisplayVersRDC:=FALSE;
		DisplayVersET1:=FALSE;
		DisplayVersET3:=FALSE;
		DisplayVersET2:=TRUE;
	ELSIF ETAGE_SUIVANT = 4 THEN
		FLECHE_VERS:=TRUE;
		DisplayVersRDC:=FALSE;
		DisplayVersET1:=FALSE;
		DisplayVersET2:=FALSE;
		DisplayVersET3:=TRUE;
	END_IF
ELSE
	FLECHE_VERS:=FALSE;
	DisplayVersRDC:=FALSE;
	DisplayVersET1:=FALSE;
	DisplayVersET2:=FALSE;
	DisplayVersET3:=FALSE;
END_IF

IF NOT ARRETcabRDC AND NOT ARRETcabD1 AND  NOT ARRETcabM1 AND  NOT ARRETcabD2 AND NOT ARRETcabM2 AND NOT ARRETcabET3 THEN
	IF PRDC OR PET3 THEN
		FinDefinition_SENS:=TRUE;
	END_IF
ELSE FinDefinition_SENS:=FALSE;END_IF



Afficher_Etage_Range:=FALSE;
END_FUNCTION

(* POU Fonctions_Usuelles/Voyants_boutons/Appel_Palier, ST *)
FUNCTION Appel_Palier : BOOL
VAR_INPUT
END_VAR
VAR
	TesteurLocal: BOOL;
	Operate_Monte: BOOL;
	CompteurLocal: INT;
	CompteurForLocal:INT;
	Niveau_Actuel: INT;
END_VAR
(*Cette fonction prend en charge un appel du palier
si l'ascenseur est initialisé elle renvoie l'appel palier,  enregistre la mémo et lance le clignotement*)
IF ESTINIT2  OR StanbyActive THEN
	IF PALRDCcligno THEN
		PALRDC:=TRUE;
	END_IF
	IF NOT PALRDC THEN
		VRDC:=FALSE;
	END_IF
	
	IF PALD1cligno THEN
		PALD1:=TRUE;
	END_IF
	IF PALM1cligno THEN
		PALM1:=TRUE;
	END_IF
	
	IF NOT PALD1 AND NOT PALM1 THEN
		V1:=FALSE;
	END_IF
	
	IF PALD2cligno THEN
		PALD2:=TRUE;
	END_IF
	IF PALM2cligno THEN
		PALM2:=TRUE;
		COUNTSTEP:=COUNTSTEP+1;
	END_IF
	IF NOT PALD2 AND NOT PALM2 THEN
		V2:=FALSE;
	END_IF

	IF PAL3cligno THEN
		PAL3:=TRUE;
		COUNTSTEP:=COUNTSTEP+1;
	END_IF

	IF NOT PAL3 THEN V3:=FALSE;END_IF
	IF PALRDC OR PALD1 OR PALM1 OR PALM2 OR PALD2 OR PAL3 OR CABRDC OR CABET1 OR CABET2 OR CABET3 THEN EXIT_StanbyFunc:=TRUE;
	ELSE EXIT_StanbyFunc:=FALSE; END_IF
END_IF
END_FUNCTION

(* POU Fonctions_Usuelles/Arret_Urgence, ST *)
FUNCTION Arret_Urgence : BOOL
VAR_INPUT
END_VAR
VAR
	ReinitAscenseurProcess: BOOL;
END_VAR
(* Cette fonction va lors d'une impulsion sur l'arret d'urgence, bloquer tous les mouvements des moteurs de l'ascenceur
et attendre une réponse de l'utilisateur quand à l'état de retour à la normal à adopter: reset / Reprise du dernier cycle.*) 
IF STOPbuttonVarImpuls THEN
	STOPbuttonVar:=TRUE;
	ReinitAscenseurProcess:=TRUE;
END_IF
IF STOPbuttonVar THEN
(*STOP MOTORS *)
	(*on coupe tout les moteurs en action*)
	STOPbuttonVar:=TRUE;

	IF ReinitAscenseurProcess THEN
		(*on sauvegarde l'état de la logique de l'ascenceur
			-boutons 
			-voyants
			-variable de prio
*)
		CABDsave:=CABD;
		CABMsave:=CABM;

		PALRDCsave:=PALRDC;
		PALD1save:=PALD1;
		PALM1save:=PALM1;
		PALD2save:=PALD2;
		PALM2save:=PALM2;
		PAL3save:=PAL3;

		CABRDCsave:=CABRDC;
		CABET1save:=CABET1;
		CABET2save:=CABET2;
		CABET3save:=CABET3;

		ARRETcabRDCsave:=ARRETcabRDC;
		ARRETcabM1save:=ARRETcabM1;
		ARRETcabD1save:=ARRETcabD1;
		ARRETcabM2save:=ARRETcabM2;
		ARRETcabD2save:=ARRETcabD2;
		ARRETcabET3save:=ARRETcabET3;

		PROCHAIN_ARRETsave:=PROCHAIN_ARRET;
		ETAGE_SUIVANTsave:=ETAGE_SUIVANT;

		ReinitAscenseurProcess:=FALSE;
	END_IF

	CABD:=FALSE;
	CABM:=FALSE;

	ORDC:=FALSE;
	O1:=FALSE;
	O2:=FALSE;
	O3:=FALSE;

	FRDC:=FALSE;
	F1:=FALSE;
	F2:=FALSE;
	F3:=FALSE;

	ARRETcabRDC:=FALSE;
	ARRETcabM1:=FALSE;
	ARRETcabD1:=FALSE;
	ARRETcabM2:=FALSE;
	ARRETcabD2:=FALSE;
	ARRETcabET3:=FALSE;

	PALRDC:=FALSE;
	PALD1:=FALSE;
	PALM1:=FALSE;
	PALD2:=FALSE;
	PALM2:=FALSE;
	PAL3:=FALSE;

	CABRDC:=FALSE;
	CABET1:=FALSE;
	CABET2:=FALSE;
	CABET3:=FALSE;
	AfficheBoutonsReset:=FALSE;
	(*Reprise si initiaisé*)
	IF ESTINIT2 THEN AfficheBoutonsReset2:=TRUE;END_IF

ELSE
	AfficheBoutonsReset:=TRUE;
	AfficheBoutonsReset2:=FALSE;
END_IF

(* si l'utilisateur demande un reset de l'ascenceur*)
IF BoutonResetVrai THEN
	ESTINIT2:=FALSE;
	STOPbuttonVar:=FALSE;
	BoutonResetVrai:=FALSE;
	ETAGE_SUIVANT:=1;
	PROCHAIN_ARRET:=0;

(* si l'utilisateur demande un retour au dernier état de l'ascenceur*)
ELSIF BoutonRepriseVrai THEN
	ESTINIT2:=TRUE;
	STOPbuttonVar:=FALSE;

	IF NOT PRDC AND NOT PET1 AND NOT PET2 AND NOT PET3 THEN
		CABD:=CABDsave;
		CABM:=CABMsave;
	END_IF

	PALRDC:=PALRDCsave;
	PALD1:=PALD1save;
	PALM1:=PALM1save;
	PALD2:=PALD2save;
	PALM2:=PALM2save;
	PAL3:=PAL3save;

	CABRDC:=CABRDCsave;
	CABET1:=CABET1save;
	CABET2:=CABET2save;
	CABET3:=CABET3save;

	ARRETcabRDC:=ARRETcabRDCsave;
	ARRETcabM1:=ARRETcabM1save;
	ARRETcabD1:=ARRETcabD1save;
	ARRETcabM2:=ARRETcabM2save;
	ARRETcabD2:=ARRETcabD2save;
	ARRETcabET3:=ARRETcabET3save;

	PROCHAIN_ARRET:=PROCHAIN_ARRETsave;
	ETAGE_SUIVANT:=ETAGE_SUIVANTsave;
	BoutonRepriseVrai:=FALSE;
END_IF
END_FUNCTION

(* POU Simulation_Visuelle/FX_Porte_Vitesse, ST *)
FUNCTION FX_Porte_Vitesse : REAL
VAR_INPUT
	PosXPorte: INT;
END_VAR
VAR
	VarLocalA: REAL;
	ValXLocal: REAL;
END_VAR
(*Cette fonction retourne la position X de la porte gauche en fonction de la position X de la porte droite*)
(* Elle permet une exacte synchronisation des deux portes*)
VarLocalA:=-(59.0/71.0);
ValXLocal:= INT_TO_REAL(PosXPorte);
FX_Porte_Vitesse:=(VarLocalA)*(ValXLocal);
END_FUNCTION

(* POU Simulation_Visuelle/FX_PorteD, ST *)
FUNCTION FX_PorteD : REAL
VAR_INPUT
	PosXPorte: INT;
END_VAR
VAR
	VarLocalA: REAL;
	ValXLocal: REAL;
END_VAR
(*Cette fonction retourne la position Y en fonction de l'axe X de la porte droite*)
VarLocalA:=(27.0/71.0);
ValXLocal:= INT_TO_REAL(PosXPorte);
VarLocalA:=(VarLocalA)*(ValXLocal);
FX_PorteD:=VarLocalA- 2;
END_FUNCTION

(* POU Simulation_Visuelle/FX_PorteG, ST *)
FUNCTION FX_PorteG : REAL
VAR_INPUT
	PosXPorte: REAL;
END_VAR
VAR
	VarLocalA: REAL;
END_VAR
(*Cette fonction retourne la position Y en fonction de l'axe X de la porte gauche*)
VarLocalA:=(20.0/59.0);
VarLocalA:=(VarLocalA)*(PosXPorte);
FX_PorteG:=VarLocalA +1;
END_FUNCTION

(* POU Fonctions_Usuelles/Last_Capt_Pres2, ST *)
FUNCTION Last_Capt_Pres2 : INT
VAR_INPUT
END_VAR
VAR
END_VAR
(*cette fonction se rapproche de get_floor mais elle permet d'obtenir le dernier capteur ou était l'ascenseur*)
IF PRDC=TRUE THEN Last_Capt_Pres2:=1; END_IF
IF PET1=TRUE THEN Last_Capt_Pres2:=2; END_IF
IF PET2=TRUE THEN Last_Capt_Pres2:=3; END_IF
IF PET3=TRUE THEN Last_Capt_Pres2:=4; END_IF
IF NOT PRDC AND NOT PET1 AND NOT PET2 AND NOT PET3 THEN Last_Capt_Pres2:=0;END_IF
END_FUNCTION

(* POU Priorite_Memo, ST *)
FUNCTION Priorite_Memo : BOOL
VAR_INPUT
END_VAR
VAR
	CompteurLocal: INT;
	ETAGE_GOOD: INT;
END_VAR
(*Cette fonction pour but de gérer les priorité en fonction de la mémorisation*)

(* Création d'un tableau pour la mémorisation des appels dans le sens montée*)
TableDeVeriteMontee[1]:=ARRETcabRDC;
TableDeVeriteMontee[2]:=ARRETcabM1;
TableDeVeriteMontee[3]:=ARRETcabM2;
TableDeVeriteMontee[4]:=ARRETcabET3;

(*Création d'un tableau pour a mémorisation des appels dans le sens de la descente*)
TableDeVeriteDesc[1]:=ARRETcabRDC;
TableDeVeriteDesc[2]:=ARRETcabD1;
TableDeVeriteDesc[3]:=ARRETcabD2;
TableDeVeriteDesc[4]:=ARRETcabET3;

(*Correspondance des tableaux précedent avec le numéro du bouton*)
ArretsDesc[1]:=0;(*Rez de chaussé*)
ArretsDesc[2]:=1;(*etage 1 descente*)
ArretsDesc[3]:=3;(*etage 2 descente*)
ArretsDesc[4]:=5;(*etage 3 *)

ArretsMonte[1]:=0;(*Rez de chaussé*)
ArretsMonte[2]:=2;(*etage 1 montée*)
ArretsMonte[3]:=4;(*etage 2 montée*)
ArretsMonte[4]:=5;(*etage 3 *)

IF NOT CABM AND NOT CABD AND NOT PRDC AND NOT PET1 AND NOT PET2 AND NOT PET3 THEN
	Niveau_Actuel:=Last_Capt_Pres();
ELSE
	Niveau_Actuel:= Last_Capt_Pres2();
END_IF
(*IF Ancien_Niveau <> 0 THEN Niveau_Actuel:= Ancien_Niveau;END_IF*)

(*On test si un des appels de la mémorisation est true*)
IF ARRETcabRDC OR ARRETcabD1 OR ARRETcabM1 OR ARRETcabD2 OR ARRETcabM2 OR ARRETcabET3 THEN

(*La gestion de la mémorisation suivante va retourner trois variables :
	-Le niveau de sortie du palier (1;2;3;4) 
	-Le niveau de sortie en fonction du bouton (RDC; PALD1,PALM1,PALD2,etc
	-Le sens de l'ascenseur

La gestion de la priorité se base sur le sens de l'ascenceur et le niveau auquel il se situe.
Après reflexion les fonctions sont divisés pour couvrir toutes les combinaisons possibles avec 4 CAS Classé par ordre depriorité  (Prio CAS1 > Prio CAS2 etc... :

	CAS 1 : L'étage se situe dans le bon sens et peut etre deservie ensuite (ex: PET1 + PALM2 + SENS montée -> TRUE);
	CAS 2 : L'étage se situe dans l'autre sens et l'asenceur doit changer de sens (ex: PET1 + PRDC + SENS montée -> Changement de sens puis CAS 1
	CAS 3: L'étage se situe dans le bon sens mais l'ascenceur doit effectuer un demi tour (ex PET2 + PALM2 + SENS montée -> demi tour puis desserte de l'étage
	CAS 4 :  l'étage se situe dans l'autre sens mais l'asenceur doit effectuer un demi tour pour y acceder ( ex PET1 +SENSmontée + PALD2 -> Demi tour puis changement de sens

Avec ces 4 cas nous pouvons faire face à toutes les situations et gérer les déplacements le plus fluidement possible. *)

	IF Niveau_Actuel > 0 THEN
		(*----------------------------------*)
		(* SENS -------- MONTEE*)
		(*----------------------------------*)
		IF SENS_M THEN
			(* On test l'étage le plus proche dans le bon sens*)
			FOR CompteurLocal:=4 TO Niveau_Actuel BY -1 DO
				IF TableDeVeriteMontee[CompteurLocal] THEN
					ETAGE_GOOD:= CompteurLocal;
				END_IF
			END_FOR
			IF ETAGE_GOOD<> 0 THEN ETAGE_SUIVANT:=ETAGE_GOOD;END_IF
			(*Si pas de résulats dans le sens*)
			(*Alors on teste dans l'autre sens*)
			IF ETAGE_SUIVANT = 9 THEN
				FOR CompteurLocal:=1 TO Niveau_Actuel BY 1 DO
					IF TableDeVeriteDesc[CompteurLocal] THEN
						ETAGE_SUIVANT:= CompteurLocal;
						SENS_M:=FALSE;
					END_IF
				END_FOR
			END_IF
			(*Si toujours pas de résulats dans le sens*)
			(*Alors on teste l'ancien sens mais inversé au niveau de l'étage*)
			IF ETAGE_SUIVANT = 9 THEN
				FOR CompteurLocal:=1 TO Niveau_Actuel BY 1 DO
					IF TableDeVeriteMontee[CompteurLocal] THEN
						ETAGE_SUIVANT:= CompteurLocal;
					END_IF
				END_FOR
			END_IF
			(*Si toujours pas de résulats dans le sens mais inversé*)
			(*Alors on teste l''autre sens mais inversé au niveau de l'étage*)
			IF ETAGE_SUIVANT = 9 THEN
				FOR CompteurLocal:=4 TO Niveau_Actuel BY -1 DO
					IF TableDeVeriteDesc[CompteurLocal] THEN
						ETAGE_SUIVANT:= CompteurLocal;
						SENS_M:=FALSE;
					END_IF
				END_FOR
			END_IF
		(*----------------------------------*)
		(* SENS -------- DESCENTE*)
		(*----------------------------------*)
		ELSIF NOT SENS_M THEN
			(* On test l'étage le plus proche dans le bon sens*)
			FOR CompteurLocal:=1 TO Niveau_Actuel BY 1 DO
				IF TableDeVeriteDesc[CompteurLocal] THEN
					ETAGE_GOOD:= CompteurLocal;
				END_IF
			END_FOR
			IF ETAGE_GOOD<> 0 THEN ETAGE_SUIVANT:=ETAGE_GOOD;END_IF
			(*Si pas de résulats dans le sens*)
			(*Alors on teste dans l'autre sens*)
			IF ETAGE_SUIVANT = 9 THEN
				FOR CompteurLocal:=4 TO Niveau_Actuel BY -1 DO
					IF TableDeVeriteMontee[CompteurLocal] THEN
						ETAGE_SUIVANT:= CompteurLocal;
						SENS_M:=TRUE;
					END_IF
				END_FOR
			END_IF
			(*Si toujours pas de résulats dans le sens*)
			(*Alors on teste l'ancien sens mais inversé au niveau de l'étage*)
			IF ETAGE_SUIVANT = 9 THEN
				FOR CompteurLocal:=4 TO Niveau_Actuel BY -1 DO
					IF TableDeVeriteDesc[CompteurLocal] THEN
						ETAGE_SUIVANT:= CompteurLocal;
					END_IF
				END_FOR
			END_IF
			(*Si toujours pas de résulats dans le sens mais inversé*)
			(*Alors on teste l''autre sens mais inversé au niveau de l'étage*)
			IF ETAGE_SUIVANT = 9 THEN
				FOR CompteurLocal:=1 TO Niveau_Actuel BY 1 DO
					IF TableDeVeriteMontee[CompteurLocal] THEN
						ETAGE_SUIVANT:= CompteurLocal;
						SENS_M:=TRUE;
					END_IF
				END_FOR
			END_IF
		END_IF
		(*----------------------------------------*)
		(*ASSIGNATION DU RESULTAT*)
		(*----------------------------------------*)
(*Récupération du résultat en fonction des listes prélablemen créer*)
		IF ETAGE_SUIVANT < 9 AND SENS_M THEN
			PROCHAIN_ARRET:=ArretsMonte[ETAGE_SUIVANT];
		ELSIF ETAGE_SUIVANT < 9 AND NOT SENS_M THEN
			PROCHAIN_ARRET:=ArretsDesc[ETAGE_SUIVANT];
		END_IF
	END_IF
END_IF
END_FUNCTION

(* POU Fonctions_Usuelles/Voyants_boutons/Quel_Etage, ST *)
FUNCTION Quel_Etage : BOOL
VAR_INPUT
END_VAR
VAR
END_VAR
(*Cette fonction permet d'activer et de désactiver les voyant de présence à l'érage en fonction des capteurs de présence*)
IF PRDC THEN
	VPALRDC:=TRUE;
	VPAL1:=FALSE;
	VPAL2:=FALSE;
	VPAL3:=FALSE;
ELSE IF PET1 THEN
	VPALRDC:=FALSE;
	VPAL1:=TRUE;
	VPAL2:=FALSE;
	VPAL3:=FALSE;
ELSE IF PET2 THEN
	VPALRDC:=FALSE;
	VPAL1:=FALSE;
	VPAL2:=TRUE;
	VPAL3:=FALSE;
ELSE IF PET3 THEN
	VPALRDC:=FALSE;
	VPAL1:=FALSE;
	VPAL2:=FALSE;
	VPAL3:=TRUE;
END_IF
END_IF
END_IF
END_IF
Quel_Etage:=TRUE;
END_FUNCTION

(* POU Fonctions_Usuelles/Capteurs/Re_ouverture, ST *)
FUNCTION Re_ouverture : BOOL
VAR_INPUT
END_VAR
VAR
END_VAR
(* Cette fonction renvoie une variable permettant la ré-ouverture d'une porte en cas d'appuis cabine ou palier*)

IF (PALRDC OR CABRDC) AND PRDC THEN
	RE_OUVRE:=TRUE;
	PALRDC:=FALSE;
	CABRDC:=FALSE;
ELSIF  (PALD1 OR CABET1)  AND PET1 AND NOT SENS_M THEN
	RE_OUVRE:=TRUE;
	PALD1:=FALSE;
	CABET1:=FALSE;
ELSIF (PALM1 OR CABET1) AND PET1 AND SENS_M THEN
	RE_OUVRE:=TRUE;
	PALM1:=FALSE;
	CABET1:=FALSE;
ELSIF (PALD2 OR CABET2) AND PET2 AND NOT SENS_M THEN
	RE_OUVRE:=TRUE;
	PALD2:=FALSE;
	CABET2:=FALSE;
ELSIF (PALM2 OR CABET2) AND PET2 AND SENS_M THEN
	RE_OUVRE:=TRUE;
	PALM2:=FALSE;
	CABET2:=FALSE;
ELSIF (PAL3 OR CABET3) AND PET3 THEN
	RE_OUVRE:=TRUE;
	PAL3:=FALSE;
	CABET3:=FALSE;
ELSE
	RE_OUVRE:=FALSE;
END_IF
IF ReOuvreCabine THEN
	RE_OUVRE:=TRUE;
END_IF
END_FUNCTION

(* POU Fonctions_Usuelles/Voyants_boutons/Reset_Arrets_CAB, ST *)
FUNCTION Reset_Arrets_CAB : BOOL
VAR_INPUT
	ARRET_EN_COURS: INT;
END_VAR
VAR
END_VAR
(* cette fonction permet de réinitialiser les boutons d'appels cabine de l'ascenceur *)
IF ARRET_EN_COURS=0 THEN
	CABRDC:=FALSE;
ELSIF ARRET_EN_COURS=1 OR ARRET_EN_COURS=2 THEN
	IF ARRET_EN_COURS = 1 THEN PALD1:=FALSE;
	ELSE PALM1:=FALSE;END_IF
	CABET1:=FALSE;
ELSIF ARRET_EN_COURS=3 OR ARRET_EN_COURS= 4 THEN
	IF ARRET_EN_COURS = 3 THEN PALD2:=FALSE;
	ELSE PALM2:=FALSE;END_IF
	CABET2:=FALSE;
ELSIF ARRET_EN_COURS=5 THEN
	CABET3:=FALSE;
END_IF
END_FUNCTION

(* POU Fonctions_Usuelles/STOP_PORTES, ST *)
FUNCTION STOP_PORTES : BOOL
VAR_INPUT
END_VAR
VAR
END_VAR
(*Cette fonction est une sécurité qui bloque l'ascenseur tant que toutes les portes ne sont pas fermé*)
IF CABD OR CABM THEN
	IF NOT PRDCfer OR NOT P1fer OR NOT P2fer OR NOT P3fer THEN
		CABDstatus:= CABD;
		CABMstatus:= CABM;
		CABD:=FALSE;
		CABM:=FALSE;
	END_IF
ELSIF NOT CABD AND NOT CABM THEN
	IF PRDCfer AND P1fer AND P2fer AND P3fer THEN
		IF CABDstatus OR CABDstatus THEN
			CABD:= CABDstatus;
			CABM:= CABMstatus;
			CABDstatus:=FALSE;
			CABMstatus:=FALSE;
		END_IF
	END_IF
END_IF
END_FUNCTION

(* POU Simulation_Visuelle/VisuCabine, ST *)
FUNCTION VisuCabine : BOOL
VAR_INPUT
END_VAR
VAR
	TimerDeTempo: TP;
	CompteurPortesVisu: INT;
	CompteurVarVisu: INT;
	CompteurDeTemps: INT;
	Step: INT;
	CompteurLocal: INT;
	ListePresence: ARRAY [1..4] OF BOOL;
	ListePosCab: ARRAY [1..9,1..2] OF INT;
	ListePresenceET: ARRAY [1..9] OF BOOL;
	MoveSlowCab: INT;
	MoveMediumCab: INT;
	MoveFastCab: INT;
END_VAR
(* Cette fonction a pour but de  faire bouger la cabine en fonction de l'activation des moteurs*)

(* La cabine enclenchera les capteurs de fin de courses si elle se trouve a la position de l'etage défini*)

(* IL y a 3 variable de vitesse défini sur 3 zones pour que la cabine se posiitonne parfaitement à l'étage et sans le dépasser*)

(*VAleurs d'initialisation du visuel*)
ListePresenceET[9]:=FALSE;

(* variable de la zone de ralentissement/ accélérationde la cabine*)
ListePosCab[9,1]:= 130 ;
ListePosCab[9,2]:= 90;

ListePosCab[1,1]:=  130;
ListePosCab[1,2]:= 90;
ListePosCab[2,1]:=  20;
ListePosCab[2,2]:= -20;
ListePosCab[3,1]:= - 90;
ListePosCab[3,2]:= - 130;
ListePosCab[4,1]:= - 200;
ListePosCab[4,2]:= - 240;

ListePresenceET[1]:=PRDC;
ListePresenceET[2]:=PET1;
ListePresenceET[3]:=PET2;
ListePresenceET[4]:=PET3;

(*La variable ZoneDepCab Zone de Départ Cabine sert au départ lent de la cabine*)
IF ZoneDepCab = 0 THEN ZoneDepCab:= 2;END_IF

IF NOT ListePresenceET[ETAGE_SUIVANT] THEN
	IF CABD THEN
		MoveSlowCab:=1;
		MoveMediumCab:=5;
		MoveFastCab:=10;
	ELSIF CABM THEN
		MoveSlowCab:=-1;
		MoveMediumCab:=-5;
		MoveFastCab:=-10;
	END_IF
	IF CABD OR CABM THEN
		wait(IN:=TRUE, PT:=T#10ms);
		IF NOT wait.Q THEN
			IF ZoneDepCab <> ETAGE_SUIVANT THEN
				IF CABmoveY > ListePosCab[ZoneDepCab,2] AND CABmoveY < ListePosCab[ZoneDepCab,1] THEN
					wait(IN:=FALSE);
					CABmoveY:=CABmoveY+MoveMediumCab;
				END_IF
			END_IF
			IF CABmoveY > ListePosCab[ETAGE_SUIVANT,2] AND CABmoveY < ListePosCab[ETAGE_SUIVANT,1] THEN
				wait(IN:=FALSE);
				CABmoveY:=CABmoveY+MoveSlowCab;

			ELSIF CABmoveY > ListePosCab[ETAGE_SUIVANT,2] -20 AND  CABmoveY <= ListePosCab[ETAGE_SUIVANT,2]  OR CABmoveY < ListePosCab[ETAGE_SUIVANT,1]+20 AND CABmoveY >= ListePosCab[ETAGE_SUIVANT,1] THEN
				wait(IN:=FALSE);
				CABmoveY:=CABmoveY+MoveMediumCab;
			ELSE
				wait(IN:=FALSE);
				CABmoveY:=CABmoveY+MoveFastCab;
			END_IF
		END_IF
	END_IF
END_IF

IF CABmoveY = 110 THEN
	PRDC:=TRUE;
	ZoneDepCab:=1;
ELSE PRDC:=FALSE;END_IF

IF CABmoveY = 0 THEN
	 PET1:=TRUE;
	IF F1 THEN ZoneDepCab:=2;END_IF
ELSE PET1:=FALSE;END_IF

IF CABmoveY = -110 THEN
	PET2:=TRUE;
	IF F2 THEN ZoneDepCab:=3;END_IF
ELSE PET2:=FALSE;END_IF

IF CABmoveY = -220 THEN
	PET3:=TRUE;
	IF F3 THEN ZoneDepCab:=4;END_IF
ELSE PET3:=FALSE;END_IF
END_FUNCTION

(* POU Simulation_Visuelle/VisuPortesET1, ST *)
FUNCTION VisuPortesET1 : BOOL
VAR_INPUT
END_VAR
VAR
	TimerDeTempo: TP;
	CompteurPortesVisu: INT;
	CompteurVarVisu: INT;
	CompteurDeTemps: INT;
	Step: INT;
	CompteurLocal: INT;
	CONTACTEUR_SEC: INT;
END_VAR
(* Cette fonction sert à fermer les portes de l'etage 1 en fonction des donné transmises par le porgramme principal*

	La fonction va simuler une fermeture sur action d'un moteur, et simuler le capteur  lorsque la coordonée de position fermé est atteinte : x=0 et y=-2*)
IF F1 OR O1 THEN
	(*On simule la position physique du contacteur avec des coordonnées*)
	IF F1 THEN CONTACTEUR_SEC:=-71;
	ELSE CONTACTEUR_SEC:=0;END_IF
	wait(IN:=TRUE, PT:=T#1ms);
	FOR CompteurLocal:=1 TO 3 BY 1 DO
		IF NOT wait.Q THEN
			wait(IN:=FALSE);
			(* en fonction de l'état du contacteur nous allons
			simuler une ouverture/fermeture de la porte*)

			(* nous allons utiliser les fonctions de coordonnées
			pour que la simulation suivent une trajectoire excate et soienet parfaitement synchronisé*)
			IF VisuET1Dx > CONTACTEUR_SEC THEN
				VisuET1Dx:=VisuET1Dx-1;
				VisuET1Dy:=FX_PorteD(VisuET1Dx);
				VisuET1Gx:=FX_Porte_Vitesse(VisuET1Dx);
				VisuET1Gy:=FX_PorteG(VisuET1Gx);
			ELSIF  VisuET1Dx < CONTACTEUR_SEC THEN
				VisuET1Dx:=VisuET1Dx+1;
				VisuET1Dy:=FX_PorteD(VisuET1Dx);
				VisuET1Gx:=FX_Porte_Vitesse(VisuET1Dx);
				VisuET1Gy:=FX_PorteG(VisuET1Gx);
			END_IF
		END_IF
	END_FOR
END_IF

IF VisuET1Dx = - 71  THEN P1fer:=TRUE;
ELSE P1fer:=FALSE;END_IF

IF VisuET1Dx = 0  THEN P1ouv:=TRUE;
ELSE P1ouv:=FALSE;END_IF
END_FUNCTION

(* POU Simulation_Visuelle/VisuPortesET2, ST *)
FUNCTION VisuPortesET2 : BOOL
VAR_INPUT
END_VAR
VAR
	TimerDeTempo: TP;
	CompteurPortesVisu: INT;
	CompteurVarVisu: INT;
	CompteurDeTemps: INT;
	Step: INT;
	CompteurLocal: INT;
	CONTACTEUR_SEC: INT;
END_VAR
(* Cette fonction sert à fermer les portes de l'etage 2 en fonction des donné transmises par le porgramme principal*

	La fonction va simuler une fermeture sur action d'un moteur, et simuler le capteur  lorsque la coordonée de position fermé est atteinte : x=0 et y=-2*)
IF F2 OR O2 THEN
	(*On simule la position physique du contacteur avec des coordonnées*)
	IF F2 THEN CONTACTEUR_SEC:=-71;
	ELSE CONTACTEUR_SEC:=0;END_IF
	wait(IN:=TRUE, PT:=T#1ms);
	FOR CompteurLocal:=1 TO 3 BY 1 DO
		IF NOT wait.Q THEN
			wait(IN:=FALSE);
			(* en fonction de l'état du contacteur nous allons
			simuler une ouverture/fermeture de la porte*)

			(* nous allons utiliser les fonctions de coordonnées
			pour que la simulation suivent une trajectoire excate et soienet parfaitement synchronisé*)
			IF VisuET2Dx > CONTACTEUR_SEC THEN
				VisuET2Dx:=VisuET2Dx-1;
				VisuET2Dy:=FX_PorteD(VisuET2Dx);
				VisuET2Gx:=FX_Porte_Vitesse(VisuET2Dx);
				VisuET2Gy:=FX_PorteG(VisuET2Gx);
			ELSIF  VisuET2Dx < CONTACTEUR_SEC THEN
				VisuET2Dx:=VisuET2Dx+1;
				VisuET2Dy:=FX_PorteD(VisuET2Dx);
				VisuET2Gx:=FX_Porte_Vitesse(VisuET2Dx);
				VisuET2Gy:=FX_PorteG(VisuET2Gx);
			END_IF
		END_IF
	END_FOR
END_IF

IF VisuET2Dx = - 71  THEN P2fer:=TRUE;
ELSE P2fer:=FALSE;END_IF

IF VisuET2Dx = 0  THEN P2ouv:=TRUE;
ELSE P2ouv:=FALSE;END_IF
END_FUNCTION

(* POU Simulation_Visuelle/VisuPortesET3, ST *)
FUNCTION VisuPortesET3 : BOOL
VAR_INPUT
END_VAR
VAR
	TimerDeTempo: TP;
	CompteurPortesVisu: INT;
	CompteurVarVisu: INT;
	CompteurDeTemps: INT;
	Step: INT;
	CompteurLocal: INT;
	CONTACTEUR_SEC: INT;
END_VAR
(* Cette fonction sert à fermer les portes de l'etage 3 en fonction des donné transmises par le porgramme principal*

	La fonction va simuler une fermeture sur action d'un moteur, et simuler le capteur  lorsque la coordonée de position fermé est atteinte : x=0 et y=-2*)
IF F3 OR O3 THEN
	(*On simule la position physique du contacteur avec des coordonnées*)
	IF F3 THEN CONTACTEUR_SEC:=-71;
	ELSE CONTACTEUR_SEC:=0;END_IF
	wait(IN:=TRUE, PT:=T#1ms);
	FOR CompteurLocal:=1 TO 3 BY 1 DO
		IF NOT wait.Q THEN
			wait(IN:=FALSE);
			(* en fonction de l'état du contacteur nous allons
			simuler une ouverture/fermeture de la porte*)

			(* nous allons utiliser les fonctions de coordonnées
			pour que la simulation suivent une trajectoire excate et soienet parfaitement synchronisé*)
			IF VisuET3Dx > CONTACTEUR_SEC THEN
				VisuET3Dx:=VisuET3Dx-1;
				VisuET3Dy:=FX_PorteD(VisuET3Dx);
				VisuET3Gx:=FX_Porte_Vitesse(VisuET3Dx);
				VisuET3Gy:=FX_PorteG(VisuET3Gx);
			ELSIF  VisuET3Dx < CONTACTEUR_SEC THEN
				VisuET3Dx:=VisuET3Dx+1;
				VisuET3Dy:=FX_PorteD(VisuET3Dx);
				VisuET3Gx:=FX_Porte_Vitesse(VisuET3Dx);
				VisuET3Gy:=FX_PorteG(VisuET3Gx);
			END_IF
		END_IF
	END_FOR
END_IF

IF VisuET3Dx = - 71  THEN P3fer:=TRUE;
ELSE P3fer:=FALSE;END_IF

IF VisuET3Dx = 0  THEN P3ouv:=TRUE;
ELSE P3ouv:=FALSE;END_IF
END_FUNCTION

(* POU Simulation_Visuelle/VisuPortesRDC, ST *)
FUNCTION VisuPortesRDC : BOOL
VAR_INPUT
END_VAR
VAR
	TimerDeTempo: TP;
	CompteurPortesVisu: INT;
	CompteurVarVisu: INT;
	CompteurDeTemps: INT;
	Step: INT;
	CompteurLocal: INT;
	CONTACTEUR_SEC: INT;
END_VAR
(* Cette fonction sert à fermer les portes du rez de chaussé en fonction des donné transmises par le porgramme principal*

	La fonction va simuler une fermeture sur action d'un moteur, et simuler le capteur  lorsque la coordonée de position fermé est atteinte : x=0 et y=-2*)
IF FRDC OR ORDC THEN
	(*On simule la position physique du contacteur avec des coordonnées*)
	IF FRDC THEN CONTACTEUR_SEC:=-71;
	ELSE CONTACTEUR_SEC:=0;END_IF
	wait(IN:=TRUE, PT:=T#1ms);
	FOR CompteurLocal:=1 TO 3 BY 1 DO
		IF NOT wait.Q THEN
			wait(IN:=FALSE);
			(* en fonction de l'état du contacteur nous allons
			simuler une ouverture/fermeture de la porte*)

			(* nous allons utiliser les fonctions de coordonnées
			pour que la simulation suivent une trajectoire excate et soienet parfaitement synchronisé*)
			IF VisuRDCDx > CONTACTEUR_SEC THEN
				VisuRDCDx:=VisuRDCDx-1;
				VisuRDCDy:=FX_PorteD(VisuRDCDx);
				VisuRDCGx:=FX_Porte_Vitesse(VisuRDCDx);
				VisuRDCGy:=FX_PorteG(VisuRDCGx);
			ELSIF  VisuRDCDx < CONTACTEUR_SEC THEN
				VisuRDCDx:=VisuRDCDx+1;
				VisuRDCDy:=FX_PorteD(VisuRDCDx);
				VisuRDCGx:=FX_Porte_Vitesse(VisuRDCDx);
				VisuRDCGy:=FX_PorteG(VisuRDCGx);
			END_IF
		END_IF
	END_FOR
END_IF

IF VisuRDCDx = - 71  THEN PRDCfer:=TRUE;
ELSE PRDCfer:=FALSE;END_IF

IF VisuRDCDx = 0  THEN PRDCouv:=TRUE;
ELSE PRDCouv:=FALSE;END_IF
END_FUNCTION

(* POU ZAuto_RUN, ST *)
  FUNCTION ZAuto_RUN : BOOL
VAR_INPUT
END_VAR
VAR
	TimerCab:TP;
	TimerPortes: TP;
END_VAR
(*Cette fonction permet de faire fonctionner les moteurs de la simulation*)

(* Init Porte*)
IF NOT InitPortesAscSalon THEN
	(*Fermeture des portes
et Instanciation d'un offset pour aligner le compteur d'étage visuel*)
	VisuRDCDx:=-60;
	VisuRDCDy:=FX_PorteD(VisuRDCDx);
	VisuRDCGx:=FX_Porte_Vitesse(VisuRDCDx);
	VisuRDCGy:=FX_PorteG(VisuRDCGx);

	VisuET1Dx:=-60;
	VisuET1Dy:=FX_PorteD(VisuET1Dx);
	VisuET1Gx:=FX_Porte_Vitesse(VisuET1Dx);
	VisuET1Gy:=FX_PorteG(VisuET1Gx);

	VisuET2Dx:=-60;
	VisuET2Dy:=FX_PorteD(VisuET2Dx);
	VisuET2Gx:=FX_Porte_Vitesse(VisuET2Dx);
	VisuET2Gy:=FX_PorteG(VisuET2Gx);

	VisuET3Dx:=-60;
	VisuET3Dy:=FX_PorteD(VisuET3Dx);
	VisuET3Gx:=FX_Porte_Vitesse(VisuET3Dx);
	VisuET3Gy:=FX_PorteG(VisuET3Gx);

	InitPortesAscSalon:=TRUE;
	DisplayNumbET1:=TRUE;
	Offset_ChiffreY:=-5;
END_IF
(*Affichage du compteur d'étage visuel*)
Afficher_Etage_Range();

(*Appel des fonctions de mouvement en focntion des moteurs*)
IF FRDC OR ORDC THEN VisuPortesRDC();END_IF
IF F1 OR O1 THEN VisuPortesET1();END_IF
IF F2 OR O2 THEN VisuPortesET2();END_IF
IF F3 OR O3 THEN VisuPortesET3();END_IF
IF CABD OR CABM THEN VisuCabine();END_IF
END_FUNCTION

(* Visualisation Visu
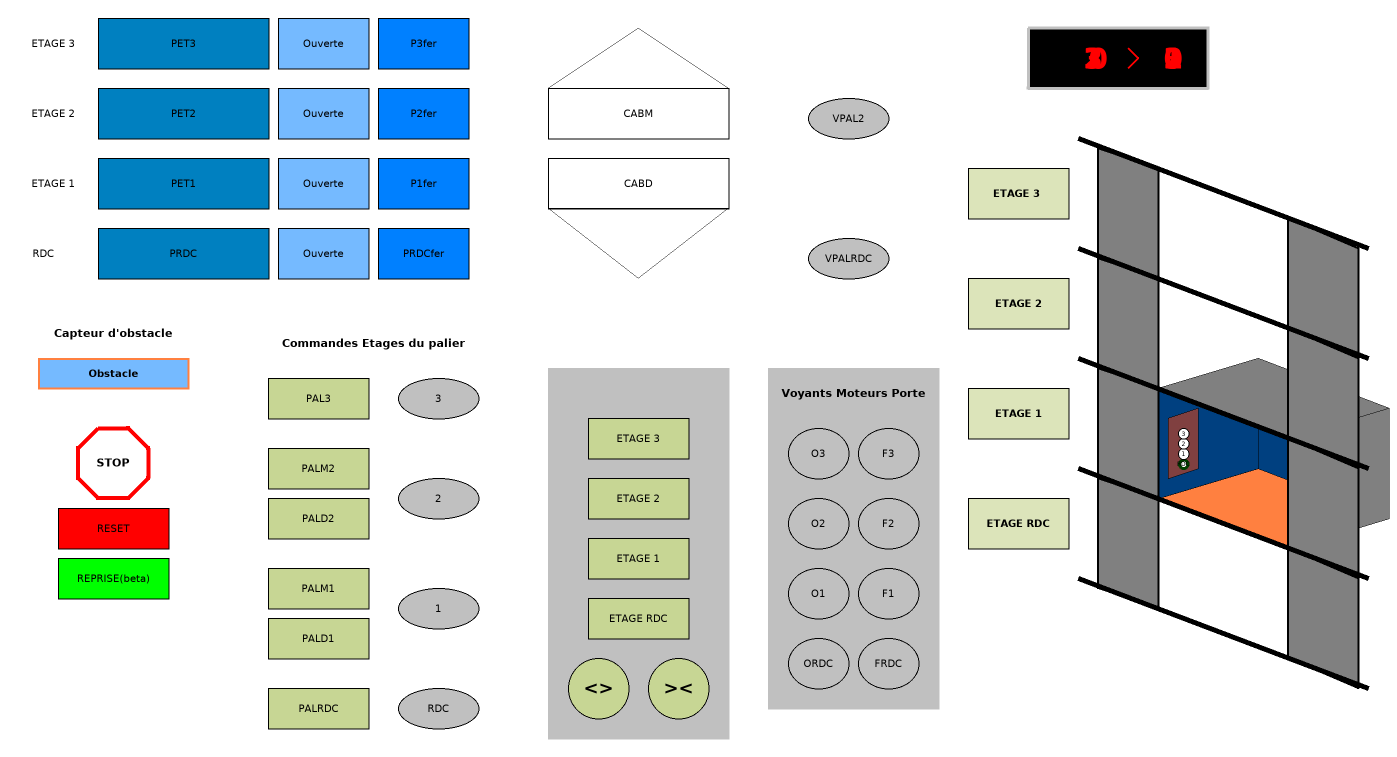
group at (1190,370)-(1421,561)
  ellipse at (20,100)-(31,111): text "RDC"; alarm colour if .CABRDC
  ellipse at (20,90)-(31,101): text "1"; alarm colour if .CABET1
  ellipse at (20,80)-(31,91): text "2"; alarm colour if .CABET2
  ellipse at (20,70)-(31,81): text "3"; alarm colour if .CABET3
ellipse at (890,440)-(951,491): text "F3"; alarm colour if .F3
rounded rectangle at (410,30)-(501,81): text "P3fer"; alarm colour if .P3fer; toggles .P3fer
rounded rectangle at (410,100)-(501,151): text "P2fer"; alarm colour if .P2fer; toggles .P2fer
rounded rectangle at (410,170)-(501,221): text "P1fer"; alarm colour if .P1fer; toggles .P1fer
rounded rectangle at (410,240)-(501,291): text "PRDCfer"; alarm colour if .PRDCfer; toggles .PRDCfer
ellipse at (820,440)-(881,491): text "O3"; alarm colour if .O3
ellipse at (820,510)-(881,561): text "O2"; alarm colour if .O2
ellipse at (820,580)-(881,631): text "O1"; alarm colour if .O1
ellipse at (820,650)-(881,701): text "ORDC"; alarm colour if .ORDC
rectangle at (580,170)-(761,221): text "CABD"; alarm colour if .CABD
rectangle at (130,240)-(301,291): text "PRDC"; alarm colour if .PRDC; toggles .PRDC
ellipse at (890,510)-(951,561): text "F2"; alarm colour if .F2
ellipse at (890,580)-(951,631): text "F1"; alarm colour if .F1
ellipse at (890,650)-(951,701): text "FRDC"; alarm colour if .FRDC; toggles .PRDCfer
rectangle at (300,330)-(511,381): text "Commandes Etages du palier"
rectangle at (20,100)-(151,151): text "ETAGE 2"
rectangle at (20,170)-(151,221): text "ETAGE 1"
rectangle at (10,240)-(141,291): text "RDC"
rounded rectangle at (310,170)-(401,221): text "Ouverte"; alarm colour if .P1ouv; toggles .P1ouv; taps .P1fer; runs Switch_ET1(PRG)
rounded rectangle at (310,240)-(401,291): text "Ouverte"; alarm colour if .PRDCouv; toggles .PRDCouv
rectangle at (130,170)-(301,221): text "PET1"; alarm colour if .PET1; toggles .PET1
rectangle at (130,100)-(301,151): text "PET2"; alarm colour if .PET2; toggles .PET2
rectangle at (130,30)-(301,81): text "PET3"; alarm colour if .PET3; toggles .PET3
rectangle at (20,30)-(151,81): text "ETAGE 3"
rounded rectangle at (300,700)-(401,741): text "PALRDC"; alarm colour if .PALRDC; taps .PALRDCcligno
rounded rectangle at (300,630)-(401,671): text "PALD1"; alarm colour if .PALD1; taps .PALD1cligno
rounded rectangle at (300,580)-(401,621): text "PALM1"; alarm colour if .PALM1; taps .PALM1cligno
rounded rectangle at (300,510)-(401,551): text "PALD2"; alarm colour if .PALD2; taps .PALD2cligno
rounded rectangle at (300,460)-(401,501): text "PALM2"; alarm colour if .PALM2; taps .PALM2cligno
rounded rectangle at (300,390)-(401,431): text "PAL3"; alarm colour if .PAL3; taps .PAL3cligno
rectangle at (580,100)-(761,151): text "CABM"; alarm colour if .CABM
ellipse at (840,40)-(921,81): text "VPAL3"; alarm colour if .VPAL3
ellipse at (840,110)-(921,151): text "VPAL2"; alarm colour if .VPAL2
ellipse at (840,180)-(921,221): text "VPAL1"; alarm colour if .VPAL1
ellipse at (840,250)-(921,291): text "VPALRDC"; alarm colour if .VPALRDC
rectangle at (40,320)-(251,371): text "Capteur d'obstacle"
polygon at (580,220)-(760,290): alarm colour if .CABD
polygon at (580,40)-(760,100): alarm colour if .CABM
rounded rectangle at (310,100)-(401,151): text "Ouverte"; alarm colour if .P2ouv; toggles .P2ouv; taps .P1fer; runs Switch_ET1(PRG)
rounded rectangle at (310,30)-(401,81): text "Ouverte"; alarm colour if .P3ouv; toggles .P3ouv; taps .P1fer; runs Switch_ET1(PRG)
polygon at (110,440)-(180,510): text "STOP"; alarm colour if .STOPbuttonVar; taps STOPbuttonVarImpuls
rounded rectangle at (70,370)-(221,401): text "Obstacle"; alarm colour if .Obs; toggles .Obs
rectangle at (820,290)-(951,341): text "Voyants Etages"
rectangle at (780,380)-(991,431): text "Voyants Moteurs Porte"
ellipse at (430,390)-(511,431): text "3"; alarm colour if .V3
ellipse at (430,490)-(511,531): text "2"; alarm colour if .V2
ellipse at (430,600)-(511,641): text "1"; alarm colour if .V1
ellipse at (430,700)-(511,741): text "RDC"; alarm colour if .VRDC
rectangle at (570,380)-(781,431): text "Commandes Cabine"
rounded rectangle at (620,430)-(721,471): text "ETAGE 3"; alarm colour if .CABET3; taps .CABET3switch
rounded rectangle at (620,490)-(721,531): text "ETAGE 2"; alarm colour if .CABET2; taps .CABET2switch
rounded rectangle at (620,550)-(721,591): text "ETAGE 1"; alarm colour if .CABET1; taps .CABET1switch
rounded rectangle at (620,610)-(721,651): text "ETAGE RDC"; alarm colour if .CABRDC; taps .CABRDCswitch
polygon at (1130,490)-(1190,620): x offset .VisuRDCGx; y offset .VisuRDCGy
polygon at (1320,560)-(1390,700): x offset .VisuRDCDx; y offset .VisuRDCDy
polygon at (1130,380)-(1190,510): x offset .VisuET1Gx; y offset .VisuET1Gy
polygon at (1320,450)-(1390,590): x offset .VisuET1Dx; y offset .VisuET1Dy
polygon at (1130,270)-(1190,400): x offset .VisuET2Gx; y offset .VisuET2Gy
polygon at (1320,340)-(1390,480): x offset .VisuET2Dx; y offset .VisuET2Dy
polygon at (1130,160)-(1190,290): x offset .VisuET3Gx; y offset .VisuET3Gy
polygon at (1320,230)-(1390,370): x offset .VisuET3Dx; y offset .VisuET3Dy
rectangle at (1000,510)-(1101,561): text "ETAGE RDC"; alarm colour if .DisplayNumbETRDC
rectangle at (1000,400)-(1101,451): text "ETAGE 1"; alarm colour if .DisplayNumbET1
rectangle at (1000,290)-(1101,341): text "ETAGE 2"; alarm colour if .DisplayNumbET2
rectangle at (1000,180)-(1101,231): text "ETAGE 3"; alarm colour if .DisplayNumbET3
rounded rectangle at (90,520)-(201,561): text "RESET"; invisible if .AfficheBoutonsReset; taps .BoutonResetVrai
rounded rectangle at (90,570)-(201,611): text "REPRISE(beta)"; invisible if NOT AfficheBoutonsReset2; taps .BoutonRepriseVrai
ellipse at (600,670)-(661,731): text "<>"; alarm colour if .ReOuvreCabine; taps .ReOuvreCabine
ellipse at (680,670)-(741,731): text "><"; alarm colour if .ForceFermeCabine; taps .ForceFermeCabine
polygon at (1080,60)-(1100,80): invisible if .NOT SENS_M
polygon at (1080,60)-(1100,80): invisible if .SENS_M
rectangle at (1110,50)-(1141,91): text "1"; invisible if NOT .DisplayNumbET1; y offset .Offset_ChiffreY
rectangle at (1190,50)-(1221,91): text "1"; invisible if NOT .DisplayVersET1; y offset .Offset_ChiffreY
rectangle at (1110,50)-(1141,91): text "2"; invisible if NOT .DisplayNumbET2; y offset .Offset_ChiffreY
rectangle at (1110,50)-(1141,91): text "3"; invisible if NOT .DisplayNumbET3; y offset .Offset_ChiffreY
rectangle at (1110,50)-(1151,91): text "0"; invisible if NOT .DisplayNumbETRDC; y offset .Offset_ChiffreY
rectangle at (1190,50)-(1221,91): text "2"; invisible if NOT .DisplayVersET2; y offset .Offset_ChiffreY
rectangle at (1190,50)-(1221,91): text "3"; invisible if NOT .DisplayVersET3; y offset .Offset_ChiffreY
rectangle at (1190,50)-(1221,91): text "0"; invisible if NOT .DisplayVersRDC; y offset .Offset_ChiffreY
polyline at (1160,60)-(1170,80): invisible if NOT .FLECHE_VERS
rectangle at (1080,50)-(1111,91): invisible if NOT .FinDefinition_SENS
30 more shapes without text or variables
*)
